C07285=1051.571,276.909,397.010,172.389,37.527,157.091
C07286=1051.565,276.657,397.040,172.386,37.524,157.091
C07287=1051.558,276.407,397.072,172.382,37.520,157.090
C07288=1051.551,276.156,397.102,172.380,37.518,157.089
C07289=1051.545,275.908,397.133,172.377,37.514,157.088
C07290=1051.539,275.660,397.164,172.374,37.511,157.088
C07291=1051.533,275.412,397.195,172.371,37.508,157.087
C07292=1051.526,275.164,397.225,172.368,37.504,157.086
C07293=1051.519,274.916,397.255,172.365,37.501,157.085
C07294=1051.513,274.668,397.286,172.363,37.498,157.085
C07295=1051.507,274.419,397.316,172.359,37.494,157.084
C07296=1051.500,274.172,397.347,172.357,37.491,157.083
C07297=1051.494,273.924,397.378,172.354,37.488,157.082
C07298=1051.487,273.675,397.408,172.350,37.485,157.082
C07299=1051.481,273.428,397.438,172.348,37.482,157.081
C07300=1051.474,273.179,397.469,172.345,37.478,157.080
C07301=1051.468,272.932,397.499,172.342,37.475,157.079
C07302=1051.461,272.683,397.529,172.339,37.472,157.079
C07303=1051.455,272.436,397.560,172.337,37.468,157.078
C07304=1051.449,272.187,397.590,172.333,37.465,157.077
C07305=1051.442,271.939,397.620,172.331,37.462,157.077
C07306=1051.436,271.691,397.651,172.328,37.458,157.076
C07307=1051.429,271.443,397.681,172.325,37.456,157.075
C07308=1051.423,271.195,397.711,172.322,37.452,157.074
C07309=1051.416,270.947,397.741,172.320,37.449,157.074
C07310=1051.410,270.699,397.772,172.317,37.446,157.073
C07311=1051.403,270.451,397.802,172.313,37.442,157.072
C07312=1051.397,270.203,397.832,172.311,37.439,157.071
C07313=1051.390,269.955,397.862,172.308,37.436,157.071
C07314=1051.384,269.707,397.893,172.305,37.433,157.070
C07315=1051.377,269.459,397.923,172.302,37.429,157.069
C07316=1051.371,269.210,397.952,172.300,37.427,157.069
C07317=1051.364,268.962,397.983,172.297,37.423,157.068
C07318=1051.358,268.714,398.013,172.294,37.420,157.067
C07319=1051.352,268.467,398.043,172.291,37.417,157.066
C07320=1051.346,268.218,398.073,172.289,37.413,157.066
C07321=1051.339,267.970,398.102,172.285,37.410,157.065
C07322=1051.332,267.722,398.133,172.283,37.407,157.064
C07323=1051.326,267.474,398.163,172.280,37.404,157.064
C07324=1051.319,267.226,398.193,172.278,37.400,157.063
C07325=1051.314,266.977,398.223,172.274,37.398,157.062
C07326=1051.306,266.729,398.253,172.272,37.394,157.061
C07327=1051.300,266.482,398.283,172.269,37.391,157.061
C07328=1051.294,266.232,398.313,172.267,37.388,157.060
C07329=1051.287,265.985,398.342,172.263,37.385,157.059
C07330=1051.281,265.737,398.372,172.261,37.381,157.058
C07331=1051.275,265.488,398.402,172.258,37.378,157.058
C07332=1051.268,265.241,398.432,172.256,37.375,157.057
C07333=1051.261,264.993,398.462,172.252,37.372,157.056
C07334=1051.255,264.744,398.492,172.250,37.368,157.056
C07335=1051.249,264.497,398.521,172.247,37.365,157.055
C07336=1051.242,264.248,398.551,172.244,37.362,157.054
C07337=1051.236,264.001,398.580,172.242,37.359,157.053
C07338=1051.229,263.753,398.610,172.238,37.356,157.053
C07339=1051.223,263.506,398.640,172.236,37.352,157.052
C07340=1051.216,263.258,398.669,172.233,37.349,157.051
C07341=1051.210,263.012,398.699,172.231,37.346,157.050
C07342=1051.204,262.764,398.729,172.228,37.343,157.050
C07343=1051.197,262.517,398.758,172.225,37.340,157.049
C07344=1051.191,262.269,398.788,172.222,37.336,157.048
C07345=1051.184,262.021,398.817,172.220,37.333,157.048
C07346=1051.178,261.772,398.846,172.217,37.330,157.047
C07347=1051.171,261.525,398.876,172.215,37.327,157.046
C07348=1051.165,261.277,398.905,172.211,37.324,157.046
C07349=1051.158,261.028,398.935,172.209,37.321,157.045
C07350=1051.151,260.780,398.964,172.206,37.318,157.044
C07351=1051.145,260.532,398.993,172.204,37.315,157.044
C07352=1051.138,260.283,399.023,172.201,37.311,157.043
C07353=1051.132,260.036,399.053,172.198,37.308,157.042
C07354=1051.125,259.787,399.082,172.196,37.305,157.042
C07355=1051.119,259.539,399.111,172.193,37.302,157.041
C07356=1051.112,259.291,399.141,172.191,37.299,157.040
C07357=1051.105,259.042,399.170,172.188,37.295,157.039
C07358=1051.099,258.794,399.199,172.184,37.293,157.039
C07359=1051.093,258.546,399.228,172.182,37.290,157.038
C07360=1051.086,258.298,399.257,172.179,37.286,157.037
C07361=1051.079,258.050,399.287,172.177,37.283,157.037
C07362=1051.072,257.802,399.316,172.175,37.280,157.036
C07363=1051.066,257.554,399.345,172.172,37.277,157.035
C07364=1051.059,257.305,399.374,172.170,37.274,157.035
C07365=1051.053,257.057,399.403,172.166,37.270,157.034
C07366=1051.047,256.809,399.432,172.164,37.267,157.033
C07367=1051.040,256.561,399.462,172.161,37.264,157.032
C07368=1051.033,256.312,399.492,172.159,37.261,157.032
C07369=1051.027,256.064,399.521,172.156,37.258,157.031
C07370=1051.021,255.816,399.550,172.154,37.255,157.030
C07371=1051.015,255.568,399.579,172.151,37.252,157.030
C07372=1051.008,255.319,399.608,172.148,37.249,157.029
C07373=1051.001,255.071,399.637,172.145,37.245,157.028
C07374=1050.995,254.823,399.666,172.143,37.242,157.028
C07375=1050.988,254.575,399.695,172.140,37.239,157.027
C07376=1050.982,254.327,399.724,172.138,37.236,157.026
C07377=1050.976,254.093,399.751,172.135,37.233,157.026
C07378=1050.970,253.860,399.779,172.133,37.230,157.025
C07379=1050.964,253.626,399.806,172.130,37.227,157.024
C07380=1050.958,253.392,399.833,172.128,37.223,157.023
C07381=1050.952,253.158,399.861,172.125,37.221,157.023
C07382=1050.946,252.925,399.888,172.123,37.218,157.022
C07383=1050.940,252.692,399.915,172.120,37.215,157.022
C07384=1050.934,252.458,399.943,172.118,37.212,157.021
C07385=1050.928,252.210,399.972,172.116,37.209,157.020
C07386=1050.920,251.962,400.001,172.113,37.205,157.019
C07387=1050.914,251.713,400.029,172.111,37.202,157.019
C07388=1050.908,251.465,400.058,172.108,37.199,157.018
C07389=1050.902,251.217,400.087,172.106,37.196,157.017
C07390=1050.896,250.969,400.116,172.103,37.192,157.017
C07391=1050.889,250.720,400.145,172.101,37.189,157.016
C07392=1050.883,250.472,400.174,172.098,37.186,157.015
C07393=1050.877,250.224,400.203,172.096,37.183,157.015
C07394=1050.871,249.975,400.232,172.093,37.180,157.014
C07395=1050.864,249.728,400.260,172.091,37.176,157.013
C07396=1050.858,249.479,400.289,172.088,37.174,157.013
C07397=1050.851,249.201,400.322,172.085,37.169,157.012
C07398=1050.843,248.924,400.354,172.082,37.166,157.011
C07399=1050.837,248.646,400.386,172.079,37.162,157.010
C07400=1050.830,248.368,400.418,172.077,37.159,157.009
C07401=1050.823,248.121,400.447,172.075,37.156,157.009
C07402=1050.817,247.872,400.475,172.072,37.152,157.008
C07403=1050.810,247.624,400.504,172.070,37.149,157.007
C07404=1050.804,247.376,400.533,172.067,37.146,157.006
C07405=1050.798,247.127,400.562,172.065,37.143,157.006
C07406=1050.792,246.879,400.591,172.062,37.139,157.005
C07407=1050.786,246.631,400.620,172.060,37.136,157.004
C07408=1050.779,246.382,400.647,172.057,37.133,157.004
C07409=1050.773,246.134,400.677,172.055,37.130,157.003
C07410=1050.767,245.886,400.706,172.052,37.126,157.002
C07411=1050.761,245.637,400.734,172.050,37.123,157.002
C07412=1050.754,245.389,400.762,172.047,37.120,157.001
C07413=1050.748,245.141,400.791,172.045,37.117,157.000
C07414=1050.741,244.892,400.820,172.042,37.114,157.000
C07415=1050.735,244.644,400.847,172.040,37.111,156.999
C07416=1050.729,244.396,400.876,172.037,37.108,156.998
C07417=1050.722,244.147,400.904,172.035,37.104,156.997
C07418=1050.716,243.899,400.933,172.032,37.101,156.997
C07419=1050.710,243.651,400.962,172.030,37.098,156.996
C07420=1050.703,243.403,400.990,172.027,37.095,156.995
C07421=1050.697,243.155,401.018,172.025,37.092,156.995
C07422=1050.690,242.907,401.046,172.022,37.088,156.994
C07423=1050.684,242.658,401.075,172.020,37.085,156.993
C07424=1050.678,242.409,401.103,172.017,37.082,156.993
C07425=1050.671,242.162,401.131,172.015,37.079,156.992
C07426=1050.666,241.913,401.160,172.013,37.076,156.991
C07427=1050.659,241.665,401.188,172.010,37.072,156.990
C07428=1050.653,241.416,401.217,172.008,37.069,156.990
C07429=1050.646,241.168,401.244,172.005,37.066,156.989
C07430=1050.639,240.920,401.273,172.003,37.063,156.988
C07431=1050.633,240.671,401.301,172.000,37.060,156.988
C07432=1050.626,240.423,401.329,171.999,37.056,156.987
C07433=1050.620,240.174,401.357,171.996,37.053,156.986
C07434=1050.613,239.926,401.386,171.994,37.050,156.986
C07435=1050.607,239.678,401.413,171.991,37.047,156.985
C07436=1050.601,239.429,401.442,171.989,37.044,156.984
C07437=1050.595,239.181,401.469,171.987,37.041,156.984
C07438=1050.588,238.933,401.497,171.984,37.037,156.983
C07439=1050.582,238.685,401.526,171.982,37.034,156.982
C07440=1050.575,238.436,401.554,171.979,37.031,156.982
C07441=1050.568,238.188,401.581,171.977,37.028,156.981
C07442=1050.562,237.939,401.610,171.974,37.025,156.980
C07443=1050.556,237.691,401.637,171.972,37.021,156.980
C07444=1050.549,237.442,401.665,171.969,37.018,156.979
C07445=1050.542,237.194,401.693,171.968,37.015,156.978
C07446=1050.537,236.946,401.721,171.965,37.012,156.977
C07447=1050.530,236.698,401.749,171.963,37.009,156.977
C07448=1050.523,236.449,401.777,171.961,37.006,156.976
C07449=1050.517,236.201,401.805,171.958,37.002,156.975
C07450=1050.511,235.952,401.833,171.956,36.999,156.975
C07451=1050.504,235.704,401.861,171.953,36.996,156.974
C07452=1050.497,235.455,401.888,171.951,36.993,156.973
C07453=1050.491,235.201,401.917,171.948,36.990,156.973
C07454=1050.485,234.947,401.945,171.946,36.986,156.972
C07455=1050.478,234.694,401.974,171.944,36.983,156.971
C07456=1050.472,234.439,402.003,171.942,36.980,156.971
C07457=1050.465,234.191,402.030,171.939,36.977,156.970
C07458=1050.459,233.943,402.058,171.937,36.973,156.969
C07459=1050.453,233.694,402.086,171.934,36.970,156.969
C07460=1050.447,233.446,402.114,171.932,36.967,156.968
C07461=1050.440,233.198,402.141,171.930,36.964,156.967
C07462=1050.433,232.949,402.169,171.928,36.960,156.966
C07463=1050.427,232.700,402.196,171.926,36.957,156.966
C07464=1050.422,232.452,402.224,171.923,36.954,156.965
C07465=1050.415,232.204,402.252,171.921,36.951,156.964
C07466=1050.408,231.955,402.280,171.918,36.948,156.964
C07467=1050.402,231.707,402.307,171.916,36.944,156.963
C07468=1050.395,231.458,402.335,171.913,36.941,156.962
C07469=1050.389,231.211,402.362,171.912,36.938,156.962
C07470=1050.383,230.962,402.389,171.909,36.935,156.961
C07471=1050.377,230.713,402.418,171.907,36.932,156.960
C07472=1050.371,230.465,402.445,171.904,36.928,156.960
C07473=1050.364,230.217,402.473,171.902,36.925,156.959
C07474=1050.357,229.968,402.501,171.901,36.922,156.958
C07475=1050.351,229.719,402.528,171.898,36.919,156.958
C07476=1050.345,229.471,402.555,171.896,36.916,156.957
C07477=1050.338,229.223,402.583,171.893,36.912,156.956
C07478=1050.331,228.974,402.610,171.891,36.909,156.956
C07479=1050.325,228.725,402.637,171.889,36.906,156.955
C07480=1050.319,228.478,402.665,171.887,36.903,156.954
C07481=1050.312,228.229,402.693,171.885,36.900,156.954
C07482=1050.306,227.980,402.720,171.882,36.897,156.953
C07483=1050.300,227.732,402.747,171.880,36.893,156.952
C07484=1050.293,227.483,402.774,171.877,36.890,156.951
C07485=1050.286,227.235,402.801,171.876,36.887,156.951
C07486=1050.279,226.987,402.829,171.873,36.884,156.950
C07487=1050.273,226.738,402.855,171.871,36.881,156.949
C07488=1050.267,226.490,402.883,171.868,36.877,156.949
C07489=1050.260,226.241,402.910,171.867,36.874,156.948
C07490=1050.254,225.993,402.938,171.865,36.871,156.947
C07491=1050.248,225.745,402.965,171.862,36.868,156.947
C07492=1050.241,225.496,402.992,171.860,36.865,156.946
C07493=1050.235,225.248,403.020,171.857,36.862,156.945
C07494=1050.228,224.999,403.046,171.856,36.858,156.945
C07495=1050.221,224.751,403.074,171.853,36.855,156.944
C07496=1050.216,224.502,403.100,171.851,36.852,156.943
C07497=1050.209,224.254,403.128,171.848,36.849,156.943
C07498=1050.203,224.006,403.155,171.847,36.846,156.942
C07499=1050.197,223.757,403.183,171.845,36.842,156.941
C07500=1050.190,223.508,403.210,171.842,36.839,156.941
C07501=1050.184,223.260,403.236,171.840,36.836,156.940
C07502=1050.177,223.012,403.263,171.838,36.833,156.939
C07503=1050.171,222.763,403.290,171.836,36.829,156.939
C07504=1050.164,222.515,403.318,171.833,36.826,156.938
C07505=1050.158,222.266,403.345,171.831,36.823,156.937
C07506=1050.152,222.018,403.372,171.830,36.819,156.937
C07507=1050.146,221.769,403.399,171.827,36.816,156.936
C07508=1050.139,221.521,403.425,171.825,36.813,156.935
C07509=1050.132,221.259,403.455,171.823,36.809,156.934
C07510=1050.126,220.997,403.483,171.821,36.806,156.934
C07511=1050.119,220.736,403.511,171.818,36.803,156.933
C07512=1050.113,220.474,403.540,171.816,36.799,156.932
C07513=1050.105,220.226,403.567,171.813,36.796,156.932
C07514=1050.099,219.977,403.593,171.812,36.793,156.931
C07515=1050.092,219.729,403.620,171.809,36.790,156.930
C07516=1050.087,219.480,403.646,171.807,36.787,156.930
C07517=1050.080,219.232,403.674,171.806,36.783,156.929
C07518=1050.073,218.984,403.700,171.803,36.780,156.928
C07519=1050.067,218.735,403.727,171.801,36.777,156.927
C07520=1050.060,218.486,403.754,171.798,36.774,156.927
C07521=1050.054,218.238,403.780,171.797,36.771,156.926
C07522=1050.047,217.989,403.808,171.794,36.767,156.925
C07523=1050.041,217.741,403.834,171.792,36.764,156.925
C07524=1050.035,217.492,403.861,171.791,36.760,156.924
C07525=1050.028,217.244,403.887,171.788,36.757,156.923
C07526=1050.022,216.995,403.914,171.786,36.754,156.923
C07527=1050.015,216.747,403.940,171.784,36.751,156.922
C07528=1050.009,216.498,403.967,171.782,36.748,156.921
C07529=1050.003,216.250,403.995,171.779,36.744,156.921
C07530=1049.996,216.001,404.021,171.778,36.741,156.920
C07531=1049.990,215.753,404.048,171.776,36.738,156.919
C07532=1049.983,215.504,404.074,171.773,36.735,156.919
C07533=1049.977,215.256,404.101,171.772,36.731,156.918
C07534=1049.970,215.007,404.127,171.769,36.728,156.917
C07535=1049.964,214.759,404.154,171.767,36.725,156.917
C07536=1049.958,214.510,404.180,171.765,36.722,156.916
C07537=1049.951,214.262,404.207,171.763,36.719,156.915
C07538=1049.945,214.013,404.233,171.761,36.715,156.915
C07539=1049.938,213.765,404.260,171.759,36.712,156.914
C07540=1049.932,213.516,404.287,171.757,36.708,156.913
C07541=1049.925,213.267,404.313,171.755,36.705,156.913
C07542=1049.920,213.019,404.340,171.753,36.702,156.912
C07543=1049.913,212.771,404.366,171.750,36.699,156.911
C07544=1049.907,212.522,404.393,171.749,36.695,156.910
C07545=1049.900,212.274,404.419,171.747,36.692,156.910
C07546=1049.894,212.025,404.446,171.744,36.689,156.909
C07547=1049.887,211.777,404.472,171.743,36.686,156.908
C07548=1049.881,211.528,404.499,171.740,36.682,156.908
C07549=1049.874,211.280,404.525,171.739,36.679,156.907
C07550=1049.868,211.031,404.550,171.736,36.675,156.906
C07551=1049.862,210.782,404.577,171.734,36.672,156.906
C07552=1049.855,210.534,404.603,171.733,36.669,156.905
C07553=1049.849,210.285,404.630,171.730,36.666,156.904
C07554=1049.842,210.037,404.656,171.729,36.662,156.904
C07555=1049.836,209.789,404.682,171.726,36.659,156.903
C07556=1049.830,209.539,404.709,171.724,36.656,156.902
C07557=1049.823,209.291,404.735,171.723,36.653,156.902
C07558=1049.817,209.043,404.761,171.720,36.649,156.901
C07559=1049.810,208.794,404.788,171.719,36.646,156.900
C07560=1049.804,208.546,404.814,171.716,36.643,156.899
C07561=1049.797,208.297,404.840,171.714,36.640,156.899
C07562=1049.791,208.049,404.866,171.712,36.636,156.898
C07563=1049.785,207.800,404.892,171.710,36.633,156.897
C07564=1049.778,207.551,404.919,171.709,36.629,156.897
C07565=1049.771,207.295,404.945,171.706,36.626,156.896
C07566=1049.765,207.039,404.972,171.704,36.623,156.895
C07567=1049.758,206.783,404.999,171.702,36.619,156.895
C07568=1049.752,206.527,405.026,171.700,36.616,156.894
C07569=1049.726,205.475,405.131,171.467,36.519,156.874
C07570=1049.720,205.226,405.157,171.464,36.516,156.873
C07571=1049.714,204.977,405.182,171.462,36.514,156.873
C07572=1049.707,204.729,405.207,171.460,36.512,156.872
C07573=1049.702,204.480,405.232,171.457,36.509,156.872
C07574=1049.695,204.232,405.256,171.454,36.507,156.871
C07575=1049.689,203.983,405.282,171.452,36.504,156.871
C07576=1049.683,203.734,405.306,171.449,36.501,156.870
C07577=1049.677,203.485,405.332,171.446,36.499,156.870
C07578=1049.671,203.237,405.357,171.444,36.497,156.869
C07579=1049.665,202.988,405.381,171.442,36.494,156.869
C07580=1049.659,202.739,405.407,171.438,36.492,156.868
C07581=1049.654,202.491,405.432,171.436,36.489,156.868
C07582=1049.648,202.242,405.456,171.434,36.487,156.867
C07583=1049.641,201.993,405.482,171.431,36.484,156.867
C07584=1049.636,201.744,405.506,171.428,36.482,156.866
C07585=1049.629,201.496,405.531,171.426,36.480,156.866
C07586=1049.623,201.247,405.555,171.424,36.477,156.865
C07587=1049.617,200.998,405.581,171.420,36.475,156.865
C07588=1049.610,200.749,405.605,171.418,36.472,156.864
C07589=1049.604,200.501,405.630,171.416,36.470,156.864
C07590=1049.599,200.252,405.654,171.413,36.467,156.863
C07591=1049.592,200.004,405.679,171.410,36.465,156.863
C07592=1049.586,199.755,405.704,171.408,36.463,156.862
C07593=1049.579,199.506,405.728,171.406,36.460,156.862
C07594=1049.574,199.258,405.753,171.403,36.458,156.861
C07595=1049.567,199.009,405.777,171.400,36.456,156.861
C07596=1049.561,198.760,405.802,171.398,36.454,156.861
C07597=1049.556,198.511,405.826,171.396,36.451,156.860
C07598=1049.549,198.263,405.851,171.392,36.449,156.860
C07599=1049.543,198.014,405.875,171.390,36.446,156.859
C07600=1049.537,197.765,405.899,171.388,36.444,156.859
C07601=1049.531,197.517,405.924,171.385,36.441,156.858
C07602=1049.525,197.267,405.949,171.383,36.439,156.858
C07603=1049.518,197.018,405.973,171.380,36.437,156.857
C07604=1049.512,196.771,405.998,171.378,36.435,156.857
C07605=1049.506,196.522,406.022,171.375,36.432,156.856
C07606=1049.501,196.273,406.046,171.373,36.430,156.856
C07607=1049.494,196.025,406.071,171.370,36.427,156.855
C07608=1049.488,195.775,406.096,171.367,36.425,156.855
C07609=1049.482,195.527,406.119,171.365,36.423,156.854
C07610=1049.476,195.278,406.144,171.363,36.421,156.854
C07611=1049.470,195.029,406.169,171.361,36.418,156.853
C07612=1049.464,194.781,406.193,171.357,36.416,156.853
C07613=1049.458,194.532,406.218,171.355,36.413,156.852
C07614=1049.452,194.283,406.241,171.353,36.411,156.852
C07615=1049.446,194.034,406.266,171.351,36.409,156.851
C07616=1049.439,193.786,406.291,171.348,36.407,156.851
C07617=1049.433,193.537,406.315,171.345,36.404,156.851
C07618=1049.427,193.288,406.339,171.343,36.402,156.850
C07619=1049.422,193.039,406.363,171.340,36.399,156.850
C07620=1049.415,192.790,406.387,171.338,36.397,156.849
C07621=1049.410,192.542,406.412,171.336,36.395,156.849
C07622=1049.403,192.293,406.436,171.333,36.393,156.848
C07623=1049.397,192.044,406.461,171.330,36.390,156.848
C07624=1049.391,191.796,406.485,171.328,36.388,156.847
C07625=1049.385,191.547,406.509,171.326,36.385,156.847
C07626=1049.379,191.298,406.533,171.324,36.384,156.846
C07627=1049.373,191.049,406.557,171.321,36.381,156.846
C07628=1049.368,190.801,406.582,171.318,36.379,156.846
C07629=1049.361,190.552,406.606,171.316,36.376,156.845
C07630=1049.354,190.267,406.633,171.314,36.374,156.845
C07631=1049.347,189.983,406.661,171.310,36.371,156.844
C07632=1049.341,189.699,406.688,171.308,36.368,156.843
C07633=1049.334,189.414,406.716,171.305,36.366,156.843
C07634=1049.328,189.166,406.740,171.302,36.364,156.842
C07635=1049.322,188.917,406.765,171.300,36.361,156.842
C07636=1049.316,188.669,406.788,171.298,36.359,156.842
C07637=1049.310,188.419,406.813,171.296,36.357,156.841
C07638=1049.304,188.171,406.837,171.293,36.354,156.841
C07639=1049.299,187.921,406.861,171.291,36.352,156.840
C07640=1049.292,187.673,406.884,171.289,36.350,156.840
C07641=1049.287,187.424,406.909,171.286,36.348,156.839
C07642=1049.281,187.175,406.933,171.283,36.345,156.839
C07643=1049.275,186.927,406.957,171.281,36.343,156.838
C07644=1049.269,186.678,406.981,171.279,36.340,156.838
C07645=1049.263,186.429,407.005,171.276,36.339,156.837
C07646=1049.257,186.180,407.029,171.274,36.336,156.837
C07647=1049.251,185.932,407.053,171.272,36.334,156.836
C07648=1049.246,185.683,407.076,171.270,36.331,156.836
C07649=1049.239,185.434,407.100,171.267,36.329,156.836
C07650=1049.234,185.185,407.125,171.264,36.327,156.835
C07651=1049.228,184.937,407.148,171.262,36.324,156.835
C07652=1049.222,184.688,407.173,171.260,36.322,156.834
C07653=1049.216,184.439,407.197,171.257,36.320,156.834
C07654=1049.211,184.190,407.220,171.255,36.318,156.833
C07655=1049.204,183.941,407.244,171.253,36.315,156.833
C07656=1049.198,183.693,407.268,171.251,36.313,156.832
C07657=1049.192,183.443,407.291,171.248,36.311,156.832
C07658=1049.186,183.195,407.315,171.246,36.309,156.832
C07659=1049.179,182.946,407.339,171.244,36.307,156.831
C07660=1049.173,182.697,407.362,171.241,36.305,156.831
C07661=1049.167,182.448,407.386,171.238,36.303,156.830
C07662=1049.161,182.199,407.409,171.236,36.301,156.830
C07663=1049.155,181.951,407.432,171.234,36.299,156.830
C07664=1049.148,181.702,407.456,171.232,36.296,156.829
C07665=1049.143,181.453,407.479,171.230,36.295,156.829
C07666=1049.135,181.204,407.503,171.227,36.292,156.828
C07667=1049.129,180.956,407.526,171.225,36.290,156.828
C07668=1049.123,180.707,407.550,171.223,36.288,156.828
C07669=1049.117,180.458,407.573,171.220,36.286,156.827
C07670=1049.111,180.209,407.596,171.217,36.284,156.827
C07671=1049.105,179.960,407.620,171.215,36.282,156.826
C07672=1049.099,179.711,407.643,171.213,36.280,156.826
C07673=1049.093,179.463,407.666,171.211,36.277,156.825
C07674=1049.086,179.214,407.690,171.208,36.276,156.825
C07675=1049.081,178.965,407.713,171.206,36.274,156.825
C07676=1049.074,178.716,407.737,171.204,36.271,156.824
C07677=1049.068,178.467,407.760,171.202,36.269,156.824
C07678=1049.062,178.219,407.784,171.199,36.267,156.823
C07679=1049.055,177.969,407.807,171.197,36.265,156.823
C07680=1049.049,177.720,407.830,171.195,36.263,156.822
C07681=1049.043,177.472,407.853,171.192,36.261,156.822
C07682=1049.038,177.223,407.876,171.190,36.259,156.822
C07683=1049.031,176.974,407.900,171.187,36.257,156.821
C07684=1049.025,176.725,407.923,171.185,36.255,156.821
C07685=1049.020,176.476,407.946,171.183,36.252,156.820
C07686=1049.013,176.227,407.970,171.181,36.250,156.820
C07687=1049.007,175.979,407.993,171.178,36.249,156.820
C07688=1049.000,175.731,408.016,171.176,36.246,156.819
C07689=1048.994,175.481,408.039,171.174,36.244,156.819
C07690=1048.988,175.232,408.062,171.172,36.242,156.818
C07691=1048.983,174.983,408.085,171.170,36.240,156.818
C07692=1048.977,174.735,408.109,171.167,36.238,156.818
C07693=1048.970,174.485,408.132,171.165,36.236,156.817
C07694=1048.963,174.201,408.158,171.163,36.233,156.817
C07695=1048.956,173.916,408.185,171.160,36.231,156.816
C07696=1048.950,173.631,408.212,171.157,36.229,156.816
C07697=1048.942,173.347,408.238,171.155,36.226,156.815
C07698=1048.937,173.098,408.261,171.153,36.224,156.815
C07699=1048.931,172.849,408.284,171.151,36.222,156.814
C07700=1048.925,172.600,408.307,171.148,36.220,156.814
C07701=1048.918,172.351,408.331,171.146,36.218,156.814
C07702=1048.912,172.102,408.354,171.144,36.216,156.813
C07703=1048.906,171.854,408.377,171.142,36.214,156.813
C07704=1048.901,171.605,408.399,171.139,36.212,156.812
C07705=1048.895,171.356,408.422,171.137,36.210,156.812
C07706=1048.889,171.107,408.445,171.135,36.207,156.812
C07707=1048.882,170.858,408.469,171.133,36.206,156.811
C07708=1048.876,170.609,408.492,171.131,36.203,156.811
C07709=1048.870,170.360,408.515,171.128,36.201,156.810
C07710=1048.865,170.112,408.538,171.126,36.199,156.810
C07711=1048.859,169.863,408.561,171.124,36.197,156.810
C07712=1048.853,169.614,408.584,171.122,36.195,156.809
C07713=1048.847,169.365,408.606,171.119,36.193,156.809
C07714=1048.840,169.116,408.629,171.117,36.191,156.808
C07715=1048.834,168.867,408.653,171.115,36.189,156.808
C07716=1048.829,168.618,408.676,171.113,36.187,156.807
C07717=1048.823,168.369,408.699,171.111,36.185,156.807
C07718=1048.817,168.121,408.722,171.108,36.183,156.807
C07719=1048.811,167.872,408.745,171.106,36.180,156.806
C07720=1048.805,167.623,408.767,171.104,36.179,156.806
C07721=1048.799,167.374,408.790,171.102,36.176,156.805
C07722=1048.793,167.125,408.813,171.099,36.174,156.805
C07723=1048.788,166.876,408.836,171.097,36.172,156.805
C07724=1048.782,166.627,408.859,171.095,36.170,156.804
C07725=1048.775,166.379,408.881,171.093,36.168,156.804
C07726=1048.769,166.129,408.904,171.091,36.166,156.804
C07727=1048.763,165.880,408.927,171.088,36.164,156.803
C07728=1048.758,165.632,408.950,171.086,36.162,156.803
C07729=1048.752,165.383,408.973,171.084,36.159,156.802
C07730=1048.745,165.134,408.996,171.082,36.158,156.802
C07731=1048.740,164.885,409.019,171.079,36.156,156.801
C07732=1048.734,164.636,409.041,171.077,36.153,156.801
C07733=1048.729,164.387,409.064,171.076,36.151,156.801
C07734=1048.723,164.138,409.087,171.074,36.150,156.800
C07735=1048.716,163.889,409.109,171.072,36.147,156.800
C07736=1048.711,163.640,409.132,171.069,36.145,156.799
C07737=1048.705,163.391,409.155,171.067,36.143,156.799
C07738=1048.699,163.143,409.178,171.065,36.141,156.799
C07739=1048.693,162.894,409.200,171.063,36.139,156.798
C07740=1048.687,162.644,409.222,171.060,36.137,156.798
C07741=1048.682,162.396,409.245,171.058,36.135,156.797
C07742=1048.676,162.147,409.268,171.056,36.133,156.797
C07743=1048.669,161.898,409.291,171.054,36.130,156.797
C07744=1048.664,161.650,409.313,171.053,36.129,156.796
C07745=1048.658,161.401,409.336,171.050,36.127,156.796
C07746=1048.653,161.151,409.358,171.048,36.124,156.795
C07747=1048.647,160.903,409.381,171.046,36.122,156.795
C07748=1048.641,160.654,409.404,171.044,36.120,156.795
C07749=1048.635,160.405,409.427,171.042,36.118,156.794
C07750=1048.629,160.156,409.448,171.039,36.116,156.794
C07751=1048.623,159.907,409.471,171.037,36.114,156.793
C07752=1048.617,159.658,409.494,171.035,36.113,156.793
C07753=1048.611,159.409,409.515,171.033,36.111,156.793
C07754=1048.605,159.160,409.538,171.031,36.108,156.792
C07755=1048.599,158.911,409.560,171.028,36.106,156.792
C07756=1048.593,158.662,409.583,171.027,36.105,156.792
C07757=1048.587,158.414,409.605,171.025,36.103,156.791
C07758=1048.579,158.128,409.630,171.022,36.100,156.791
C07759=1048.572,157.843,409.656,171.020,36.098,156.790
C07760=1048.565,157.558,409.681,171.017,36.096,156.790
C07761=1048.559,157.272,409.706,171.015,36.094,156.790
C07762=1048.553,157.024,409.729,171.013,36.092,156.789
C07763=1048.547,156.774,409.751,171.011,36.090,156.789
C07764=1048.541,156.525,409.774,171.008,36.088,156.788
C07765=1048.535,156.277,409.796,171.006,36.086,156.788
C07766=1048.528,156.028,409.818,171.004,36.084,156.788
C07767=1048.523,155.779,409.841,171.003,36.082,156.787
C07768=1048.517,155.530,409.863,171.001,36.080,156.787
C07769=1048.510,155.281,409.885,170.998,36.078,156.786
C07770=1048.505,155.031,409.907,170.996,36.076,156.786
C07771=1048.498,154.783,409.929,170.994,36.074,156.786
C07772=1048.492,154.534,409.951,170.992,36.072,156.785
C07773=1048.486,154.285,409.974,170.990,36.070,156.785
C07774=1048.481,154.036,409.995,170.987,36.069,156.785
C07775=1048.475,153.787,410.017,170.985,36.067,156.784
C07776=1048.468,153.539,410.039,170.984,36.064,156.784
C07777=1048.462,153.289,410.061,170.982,36.062,156.783
C07778=1048.456,153.040,410.084,170.980,36.061,156.783
C07779=1048.450,152.791,410.106,170.977,36.059,156.783
C07780=1048.444,152.542,410.127,170.975,36.057,156.782
C07781=1048.437,152.293,410.149,170.973,36.055,156.782
C07782=1048.432,152.044,410.172,170.971,36.053,156.782
C07783=1048.426,151.795,410.193,170.969,36.051,156.781
C07784=1048.420,151.547,410.215,170.968,36.049,156.781
C07785=1048.414,151.298,410.237,170.965,36.048,156.781
C07786=1048.408,151.048,410.259,170.963,36.046,156.780
C07787=1048.402,150.799,410.282,170.961,36.043,156.780
C07788=1048.396,150.550,410.303,170.959,36.041,156.779
C07789=1048.390,150.301,410.325,170.957,36.039,156.779
C07790=1048.384,150.053,410.347,170.954,36.038,156.779
C07791=1048.378,149.804,410.368,170.953,36.036,156.778
C07792=1048.372,149.554,410.391,170.951,36.034,156.778
C07793=1048.366,149.306,410.413,170.949,36.032,156.778
C07794=1048.359,149.057,410.435,170.947,36.030,156.777
C07795=1048.354,148.808,410.456,170.944,36.028,156.777
C07796=1048.348,148.559,410.478,170.942,36.026,156.777
C07797=1048.342,148.310,410.499,170.941,36.025,156.776
C07798=1048.335,148.061,410.522,170.939,36.023,156.776
C07799=1048.329,147.812,410.543,170.937,36.021,156.775
C07800=1048.324,147.562,410.565,170.935,36.019,156.775
C07801=1048.318,147.314,410.587,170.932,36.017,156.775
C07802=1048.312,147.065,410.608,170.930,36.015,156.774
C07803=1048.305,146.816,410.631,170.928,36.013,156.774
C07804=1048.299,146.567,410.652,170.927,36.012,156.774
C07805=1048.293,146.318,410.674,170.925,36.010,156.773
C07806=1048.287,146.069,410.695,170.922,36.008,156.773
C07807=1048.281,145.820,410.716,170.920,36.006,156.773
C07808=1048.274,145.571,410.738,170.918,36.004,156.772
C07809=1048.268,145.322,410.760,170.916,36.002,156.772
C07810=1048.262,145.073,410.781,170.915,36.000,156.772
C07811=1048.257,144.824,410.802,170.913,35.998,156.771
C07812=1048.250,144.575,410.824,170.910,35.997,156.771
C07813=1048.244,144.326,410.846,170.908,35.995,156.771
C07814=1048.238,144.077,410.867,170.906,35.993,156.770
C07815=1048.232,143.829,410.889,170.904,35.991,156.770
C07816=1048.226,143.580,410.911,170.903,35.989,156.769
C07817=1048.220,143.330,410.933,170.900,35.987,156.769
C07818=1048.214,143.081,410.954,170.898,35.985,156.769
C07819=1048.208,142.833,410.976,170.896,35.984,156.768
C07820=1048.202,142.583,410.997,170.894,35.982,156.768
C07821=1048.196,142.334,411.019,170.893,35.980,156.768
C07822=1048.189,142.049,411.042,170.889,35.977,156.767
C07823=1048.182,141.763,411.068,170.887,35.975,156.767
C07824=1048.175,141.477,411.092,170.885,35.974,156.766
C07825=1048.168,141.193,411.116,170.883,35.971,156.766
C07826=1048.162,140.943,411.138,170.881,35.969,156.766
C07827=1048.156,140.694,411.160,170.879,35.967,156.765
C07828=1048.150,140.446,411.181,170.877,35.966,156.765
C07829=1048.144,140.196,411.203,170.875,35.964,156.765
C07830=1048.138,139.947,411.223,170.873,35.962,156.764
C07831=1048.133,139.698,411.245,170.872,35.960,156.764
C07832=1048.126,139.449,411.266,170.870,35.958,156.764
C07833=1048.120,139.200,411.288,170.867,35.956,156.763
C07834=1048.113,138.951,411.309,170.865,35.954,156.763
C07835=1048.108,138.702,411.330,170.863,35.952,156.762
C07836=1048.102,138.453,411.352,170.862,35.951,156.762
C07837=1048.096,138.203,411.373,170.860,35.949,156.762
C07838=1048.089,137.955,411.394,170.858,35.947,156.762
C07839=1048.083,137.706,411.415,170.855,35.946,156.761
C07840=1048.077,137.457,411.437,170.853,35.944,156.761
C07841=1048.072,137.208,411.458,170.852,35.942,156.760
C07842=1048.065,136.959,411.478,170.850,35.940,156.760
C07843=1048.059,136.709,411.500,170.848,35.938,156.760
C07844=1048.053,136.461,411.521,170.845,35.936,156.759
C07845=1048.047,136.211,411.542,170.843,35.934,156.759
C07846=1048.040,135.962,411.563,170.842,35.932,156.759
C07847=1048.035,135.714,411.585,170.840,35.931,156.758
C07848=1048.029,135.464,411.606,170.838,35.929,156.758
C07849=1048.023,135.216,411.626,170.836,35.927,156.758
C07850=1048.017,134.966,411.648,170.834,35.926,156.757
C07851=1048.010,134.717,411.669,170.832,35.924,156.757
C07852=1048.004,134.468,411.689,170.830,35.922,156.757
C07853=1047.998,134.219,411.711,170.828,35.920,156.756
C07854=1047.992,133.970,411.733,170.826,35.918,156.756
C07855=1047.986,133.721,411.753,170.825,35.916,156.756
C07856=1047.980,133.472,411.774,170.822,35.914,156.755
C07857=1047.974,133.224,411.796,170.820,35.913,156.755
C07858=1047.968,132.974,411.816,170.818,35.911,156.755
C07859=1047.962,132.726,411.837,170.817,35.909,156.754
C07860=1047.956,132.476,411.859,170.815,35.907,156.754
C07861=1047.949,132.227,411.879,170.813,35.906,156.754
C07862=1047.944,131.978,411.900,170.810,35.904,156.753
C07863=1047.938,131.728,411.921,170.809,35.902,156.753
C07864=1047.932,131.480,411.942,170.807,35.900,156.753
C07865=1047.926,131.230,411.963,170.805,35.898,156.752
C07866=1047.919,130.982,411.984,170.803,35.897,156.752
C07867=1047.914,130.732,412.004,170.802,35.895,156.752
C07868=1047.907,130.484,412.025,170.799,35.893,156.751
C07869=1047.901,130.235,412.045,170.797,35.891,156.751
C07870=1047.895,129.986,412.067,170.795,35.890,156.751
C07871=1047.888,129.736,412.087,170.793,35.888,156.750
C07872=1047.883,129.487,412.109,170.792,35.886,156.750
C07873=1047.876,129.238,412.129,170.790,35.884,156.750
C07874=1047.870,128.990,412.150,170.787,35.882,156.749
C07875=1047.864,128.740,412.171,170.785,35.881,156.749
C07876=1047.857,128.491,412.192,170.784,35.879,156.749
C07877=1047.851,128.242,412.212,170.782,35.877,156.748
C07878=1047.845,127.992,412.233,170.780,35.876,156.748
C07879=1047.839,127.744,412.253,170.778,35.874,156.748
C07880=1047.832,127.495,412.274,170.776,35.872,156.747
C07881=1047.827,127.246,412.295,170.774,35.871,156.747
C07882=1047.820,126.997,412.315,170.772,35.869,156.747
C07883=1047.815,126.748,412.336,170.770,35.867,156.746
C07884=1047.808,126.499,412.357,170.769,35.866,156.746
C07885=1047.801,126.249,412.377,170.767,35.864,156.746
C07886=1047.794,125.964,412.401,170.765,35.862,156.745
C07887=1047.787,125.678,412.424,170.762,35.860,156.745
C07888=1047.781,125.392,412.447,170.760,35.857,156.745
C07889=1047.773,125.106,412.471,170.758,35.855,156.744
C07890=1047.768,124.857,412.492,170.756,35.854,156.744
C07891=1047.761,124.608,412.513,170.754,35.852,156.744
C07892=1047.755,124.359,412.533,170.752,35.850,156.743
C07893=1047.749,124.110,412.553,170.750,35.849,156.743
C07894=1047.743,123.861,412.574,170.748,35.847,156.743
C07895=1047.737,123.613,412.594,170.746,35.845,156.742
C07896=1047.731,123.363,412.615,170.745,35.844,156.742
C07897=1047.725,123.114,412.635,170.743,35.842,156.742
C07898=1047.718,122.865,412.656,170.741,35.840,156.741
C07899=1047.713,122.616,412.677,170.739,35.838,156.741
C07900=1047.706,122.366,412.697,170.737,35.837,156.741
C07901=1047.700,122.118,412.717,170.735,35.835,156.740
C07902=1047.694,121.868,412.738,170.733,35.833,156.740
C07903=1047.688,121.620,412.759,170.732,35.831,156.740
C07904=1047.682,121.371,412.779,170.730,35.829,156.739
C07905=1047.676,121.121,412.800,170.727,35.828,156.739
C07906=1047.670,120.872,412.820,170.726,35.826,156.739
C07907=1047.663,120.623,412.840,170.724,35.824,156.738
C07908=1047.658,120.374,412.861,170.722,35.822,156.738
C07909=1047.652,120.125,412.881,170.720,35.820,156.738
C07910=1047.645,119.876,412.901,170.719,35.818,156.737
C07911=1047.639,119.627,412.921,170.716,35.817,156.737
C07912=1047.633,119.377,412.942,170.714,35.815,156.737
C07913=1047.627,119.128,412.962,170.713,35.813,156.736
C07914=1047.621,118.880,412.982,170.711,35.812,156.736
C07915=1047.616,118.630,413.003,170.709,35.810,156.736
C07916=1047.609,118.382,413.024,170.708,35.808,156.736
C07917=1047.603,118.132,413.044,170.706,35.807,156.735
C07918=1047.597,117.883,413.065,170.703,35.805,156.735
C07919=1047.591,117.634,413.085,170.701,35.803,156.734
C07920=1047.585,117.385,413.105,170.700,35.801,156.734
C07921=1047.579,117.136,413.125,170.698,35.799,156.734
C07922=1047.574,116.887,413.146,170.696,35.798,156.734
C07923=1047.567,116.637,413.166,170.695,35.796,156.733
C07924=1047.561,116.388,413.186,170.692,35.794,156.733
C07925=1047.555,116.139,413.206,170.690,35.792,156.732
C07926=1047.549,115.890,413.227,170.689,35.790,156.732
C07927=1047.543,115.641,413.247,170.687,35.788,156.732
C07928=1047.537,115.392,413.267,170.685,35.787,156.732
C07929=1047.532,115.143,413.287,170.684,35.785,156.731
C07930=1047.525,114.893,413.308,170.681,35.783,156.731
C07931=1047.519,114.645,413.327,170.679,35.781,156.731
C07932=1047.513,114.396,413.347,170.678,35.780,156.730
C07933=1047.507,114.146,413.368,170.676,35.778,156.730
C07934=1047.501,113.897,413.388,170.674,35.776,156.730
C07935=1047.495,113.648,413.408,170.673,35.774,156.729
C07936=1047.489,113.399,413.429,170.670,35.773,156.729
C07937=1047.483,113.150,413.449,170.668,35.771,156.729
C07938=1047.477,112.901,413.469,170.666,35.769,156.728
C07939=1047.471,112.651,413.488,170.665,35.768,156.728
C07940=1047.465,112.402,413.508,170.663,35.766,156.728
C07941=1047.459,112.153,413.528,170.661,35.764,156.727
C07942=1047.453,111.905,413.548,170.660,35.763,156.727
C07943=1047.446,111.655,413.568,170.657,35.761,156.727
C07944=1047.440,111.406,413.588,170.655,35.759,156.726
C07945=1047.434,111.157,413.608,170.654,35.757,156.726
C07946=1047.428,110.907,413.628,170.652,35.756,156.726
C07947=1047.422,110.658,413.648,170.650,35.754,156.725
C07948=1047.416,110.410,413.668,170.649,35.752,156.725
C07949=1047.409,110.160,413.688,170.647,35.751,156.725
C07950=1047.402,109.874,413.710,170.644,35.749,156.724
C07951=1047.395,109.588,413.733,170.642,35.747,156.724
C07952=1047.388,109.303,413.756,170.640,35.745,156.724
C07953=1047.381,109.017,413.779,170.638,35.743,156.723
C07954=1047.375,108.768,413.799,170.636,35.741,156.723
C07955=1047.369,108.518,413.818,170.635,35.739,156.723
C07956=1047.363,108.269,413.838,170.632,35.738,156.723
C07957=1047.356,108.020,413.858,170.630,35.736,156.722
C07958=1047.350,107.771,413.877,170.629,35.734,156.722
C07959=1047.344,107.522,413.897,170.627,35.733,156.722
C07960=1047.338,107.273,413.917,170.625,35.731,156.721
C07961=1047.332,107.024,413.937,170.624,35.729,156.721
C07962=1047.326,106.774,413.956,170.622,35.728,156.721
C07963=1047.320,106.526,413.976,170.619,35.726,156.720
C07964=1047.313,106.276,413.995,170.618,35.724,156.720
C07965=1047.307,106.027,414.015,170.616,35.723,156.720
C07966=1047.301,105.778,414.035,170.614,35.721,156.719
C07967=1047.295,105.529,414.054,170.613,35.719,156.719
C07968=1047.289,105.280,414.074,170.611,35.718,156.719
C07969=1047.283,105.030,414.095,170.609,35.716,156.718
C07970=1047.276,104.781,414.113,170.607,35.714,156.718
C07971=1047.270,104.532,414.133,170.605,35.712,156.718
C07972=1047.265,104.283,414.153,170.603,35.711,156.718
C07973=1047.259,104.034,414.173,170.602,35.709,156.717
C07974=1047.252,103.784,414.192,170.600,35.707,156.717
C07975=1047.246,103.535,414.212,170.598,35.706,156.717
C07976=1047.239,103.287,414.231,170.597,35.704,156.716
C07977=1047.234,103.037,414.251,170.594,35.702,156.716
C07978=1047.228,102.789,414.271,170.592,35.701,156.716
C07979=1047.222,102.539,414.290,170.591,35.699,156.715
C07980=1047.216,102.290,414.310,170.589,35.697,156.715
C07981=1047.209,102.040,414.329,170.587,35.695,156.715
C07982=1047.203,101.792,414.349,170.586,35.694,156.714
C07983=1047.197,101.542,414.368,170.584,35.692,156.714
C07984=1047.191,101.293,414.388,170.582,35.690,156.714
C07985=1047.186,101.044,414.407,170.580,35.689,156.713
C07986=1047.179,100.796,414.427,170.578,35.687,156.713
C07987=1047.173,100.545,414.446,170.577,35.685,156.713
C07988=1047.167,100.297,414.466,170.575,35.684,156.713
C07989=1047.160,100.047,414.485,170.573,35.682,156.712
C07990=1047.155,99.798,414.504,170.571,35.680,156.712
C07991=1047.148,99.549,414.523,170.569,35.679,156.712
C07992=1047.142,99.300,414.543,170.567,35.677,156.711
C07993=1047.136,99.051,414.563,170.566,35.675,156.711
C07994=1047.129,98.801,414.582,170.564,35.673,156.711
C07995=1047.123,98.552,414.601,170.562,35.672,156.711
C07996=1047.117,98.303,414.620,170.561,35.670,156.710
C07997=1047.111,98.054,414.640,170.559,35.668,156.710
C07998=1047.105,97.805,414.658,170.556,35.667,156.710
C07999=1047.099,97.556,414.678,170.555,35.665,156.709
C08000=1047.092,97.306,414.698,170.553,35.664,156.709
C08001=1047.086,97.057,414.716,170.551,35.662,156.709
C08002=1047.080,96.808,414.736,170.550,35.660,156.708
C08003=1047.074,96.559,414.755,170.548,35.659,156.708
C08004=1047.068,96.309,414.774,170.546,35.657,156.708
C08005=1047.061,96.060,414.793,170.544,35.656,156.708
C08006=1047.055,95.812,414.813,170.542,35.654,156.707
C08007=1047.049,95.562,414.831,170.540,35.652,156.707
C08008=1047.043,95.313,414.851,170.539,35.651,156.707
C08009=1047.037,95.064,414.869,170.537,35.649,156.706
C08010=1047.030,94.814,414.890,170.535,35.647,156.706
C08011=1047.024,94.565,414.908,170.534,35.646,156.706
C08012=1047.018,94.316,414.928,170.531,35.644,156.705
C08013=1047.012,94.066,414.947,170.529,35.642,156.705
C08014=1047.006,93.781,414.969,170.528,35.641,156.705
C08015=1046.998,93.495,414.990,170.526,35.639,156.704
C08016=1046.991,93.209,415.013,170.524,35.637,156.704
C08017=1046.984,92.923,415.034,170.522,35.634,156.704
C08018=1046.978,92.674,415.054,170.520,35.633,156.703
C08019=1046.972,92.425,415.073,170.518,35.631,156.703
C08020=1046.966,92.176,415.092,170.516,35.630,156.703
C08021=1046.959,91.927,415.111,170.514,35.628,156.702
C08022=1046.954,91.677,415.130,170.513,35.626,156.702
C08023=1046.947,91.428,415.149,170.511,35.625,156.702
C08024=1046.942,91.179,415.168,170.509,35.623,156.702
C08025=1046.935,90.930,415.187,170.508,35.621,156.701
C08026=1046.929,90.681,415.207,170.506,35.620,156.701
C08027=1046.923,90.431,415.225,170.504,35.618,156.701
C08028=1046.917,90.182,415.245,170.502,35.616,156.700
C08029=1046.911,89.933,415.263,170.500,35.614,156.700
C08030=1046.904,89.684,415.282,170.499,35.613,156.700
C08031=1046.898,89.435,415.300,170.497,35.611,156.699
C08032=1046.892,89.185,415.320,170.495,35.609,156.699
C08033=1046.886,88.936,415.338,170.494,35.608,156.699
C08034=1046.879,88.687,415.357,170.491,35.606,156.699
C08035=1046.873,88.438,415.376,170.489,35.605,156.698
C08036=1046.867,88.188,415.395,170.488,35.603,156.698
C08037=1046.861,87.939,415.414,170.486,35.602,156.698
C08038=1046.854,87.690,415.432,170.484,35.600,156.697
C08039=1046.848,87.441,415.451,170.483,35.599,156.697
C08040=1046.842,87.192,415.470,170.481,35.597,156.697
C08041=1046.836,86.943,415.489,170.479,35.595,156.697
C08042=1046.829,86.693,415.507,170.477,35.593,156.696
C08043=1046.823,86.444,415.526,170.475,35.592,156.696
C08044=1046.817,86.195,415.545,170.473,35.590,156.696
C08045=1046.811,85.946,415.564,170.472,35.589,156.695
C08046=1046.804,85.697,415.583,170.470,35.587,156.695
C08047=1046.798,85.448,415.601,170.469,35.586,156.695
C08048=1046.792,85.198,415.619,170.467,35.584,156.695
C08049=1046.786,84.948,415.638,170.464,35.582,156.694
C08050=1046.780,84.699,415.657,170.463,35.581,156.694
C08051=1046.773,84.450,415.676,170.461,35.579,156.694
C08052=1046.767,84.201,415.694,170.459,35.578,156.693
C08053=1046.761,83.952,415.714,170.458,35.576,156.693
C08054=1046.755,83.702,415.732,170.456,35.574,156.693
C08055=1046.748,83.453,415.751,170.454,35.572,156.693
C08056=1046.743,83.204,415.768,170.453,35.571,156.692
C08057=1046.736,82.955,415.787,170.450,35.569,156.692
C08058=1046.731,82.706,415.806,170.449,35.567,156.692
C08059=1046.724,82.457,415.825,170.447,35.566,156.691
C08060=1046.718,82.207,415.844,170.445,35.564,156.691
C08061=1046.711,81.958,415.862,170.444,35.563,156.691
C08062=1046.705,81.709,415.880,170.442,35.561,156.690
C08063=1046.700,81.459,415.900,170.440,35.560,156.690
C08064=1046.693,81.210,415.918,170.439,35.558,156.690
C08065=1046.687,80.961,415.937,170.436,35.557,156.690
C08066=1046.681,80.712,415.955,170.434,35.555,156.689
C08067=1046.675,80.463,415.973,170.433,35.553,156.689
C08068=1046.669,80.213,415.992,170.431,35.551,156.689
C08069=1046.663,79.964,416.011,170.430,35.550,156.688
C08070=1046.656,79.715,416.030,170.428,35.548,156.688
C08071=1046.650,79.465,416.047,170.426,35.546,156.688
C08072=1046.644,79.216,416.066,170.425,35.544,156.687
C08073=1046.639,78.967,416.085,170.422,35.543,156.687
C08074=1046.632,78.718,416.103,170.420,35.541,156.687
C08075=1046.626,78.469,416.122,170.419,35.540,156.687
C08076=1046.620,78.219,416.140,170.417,35.538,156.686
C08077=1046.614,77.970,416.158,170.416,35.537,156.686
C08078=1046.607,77.684,416.179,170.414,35.535,156.686
C08079=1046.599,77.398,416.200,170.412,35.533,156.685
C08080=1046.593,77.112,416.222,170.409,35.531,156.685
C08081=1046.585,76.826,416.243,170.407,35.529,156.685
C08082=1046.579,76.577,416.261,170.405,35.528,156.685
C08083=1046.573,76.328,416.279,170.404,35.526,156.684
C08084=1046.566,76.079,416.298,170.402,35.525,156.684
C08085=1046.560,75.829,416.316,170.400,35.523,156.684
C08086=1046.554,75.580,416.334,170.399,35.521,156.683
C08087=1046.548,75.331,416.352,170.397,35.520,156.683
C08088=1046.541,75.081,416.371,170.396,35.518,156.683
C08089=1046.536,74.832,416.388,170.393,35.516,156.682
C08090=1046.529,74.583,416.407,170.391,35.515,156.682
C08091=1046.523,74.334,416.426,170.390,35.513,156.682
C08092=1046.517,74.084,416.444,170.388,35.512,156.682
C08093=1046.510,73.836,416.462,170.386,35.511,156.681
C08094=1046.503,73.586,416.480,170.385,35.509,156.681
C08095=1046.498,73.337,416.498,170.383,35.507,156.681
C08096=1046.492,73.088,416.516,170.381,35.505,156.681
C08097=1046.485,72.839,416.534,170.379,35.504,156.680
C08098=1046.479,72.589,416.552,170.377,35.502,156.680
C08099=1046.473,72.340,416.571,170.375,35.501,156.680
C08100=1046.467,72.091,416.589,170.374,35.499,156.679
C08101=1046.461,71.842,416.607,170.372,35.498,156.679
C08102=1046.454,71.592,416.625,170.371,35.496,156.679
C08103=1046.448,71.342,416.643,170.369,35.495,156.679
C08104=1046.442,71.094,416.661,170.367,35.493,156.678
C08105=1046.436,70.844,416.679,170.365,35.491,156.678
C08106=1046.429,70.595,416.697,170.363,35.489,156.678
C08107=1046.423,70.345,416.715,170.361,35.488,156.678
C08108=1046.417,70.097,416.734,170.360,35.486,156.677
C08109=1046.411,69.847,416.752,170.358,35.485,156.677
C08110=1046.405,69.597,416.769,170.356,35.483,156.677
C08111=1046.399,69.348,416.788,170.355,35.482,156.676
C08112=1046.392,69.100,416.805,170.353,35.480,156.676
C08113=1046.386,68.850,416.823,170.351,35.479,156.676
C08114=1046.380,68.601,416.842,170.349,35.477,156.675
C08115=1046.374,68.351,416.860,170.347,35.475,156.675
C08116=1046.367,68.102,416.877,170.346,35.474,156.675
C08117=1046.361,67.853,416.895,170.344,35.472,156.675
C08118=1046.355,67.603,416.913,170.342,35.471,156.674
C08119=1046.349,67.354,416.931,170.341,35.469,156.674
C08120=1046.342,67.106,416.949,170.339,35.468,156.674
C08121=1046.336,66.856,416.967,170.337,35.466,156.674
C08122=1046.330,66.606,416.985,170.335,35.464,156.673
C08123=1046.324,66.357,417.002,170.333,35.463,156.673
C08124=1046.317,66.108,417.020,170.331,35.461,156.673
C08125=1046.311,65.859,417.038,170.330,35.460,156.673
C08126=1046.306,65.609,417.056,170.328,35.458,156.672
C08127=1046.299,65.360,417.073,170.327,35.457,156.672
C08128=1046.292,65.111,417.092,170.325,35.455,156.672
C08129=1046.286,64.861,417.110,170.323,35.454,156.671
C08130=1046.280,64.612,417.127,170.321,35.452,156.671
C08131=1046.274,64.363,417.145,170.319,35.450,156.671
C08132=1046.268,64.113,417.163,170.317,35.449,156.671
C08133=1046.261,63.865,417.180,170.316,35.447,156.670
C08134=1046.255,63.615,417.198,170.314,35.446,156.670
C08135=1046.248,63.366,417.215,170.312,35.445,156.670
C08136=1046.242,63.116,417.233,170.311,35.443,156.670
C08137=1046.236,62.867,417.250,170.309,35.441,156.669
C08138=1046.230,62.617,417.268,170.307,35.440,156.669
C08139=1046.223,62.368,417.286,170.305,35.438,156.669
C08140=1046.217,62.119,417.303,170.303,35.437,156.669
C08141=1046.210,61.870,417.321,170.301,35.436,156.668
C08142=1046.203,61.584,417.342,170.299,35.434,156.668
C08143=1046.196,61.298,417.362,170.297,35.432,156.668
C08144=1046.189,61.012,417.381,170.296,35.430,156.667
C08145=1046.180,60.725,417.401,170.294,35.428,156.667
C08146=1046.175,60.476,417.419,170.292,35.427,156.667
C08147=1046.168,60.227,417.436,170.290,35.426,156.667
C08148=1046.162,59.977,417.454,170.288,35.424,156.666
C08149=1046.156,59.728,417.471,170.286,35.423,156.666
C08150=1046.150,59.479,417.489,170.284,35.421,156.666
C08151=1046.143,59.229,417.506,170.283,35.419,156.665
C08152=1046.136,58.981,417.523,170.281,35.418,156.665
C08153=1046.130,58.731,417.541,170.279,35.417,156.665
C08154=1046.123,58.481,417.559,170.278,35.415,156.665
C08155=1046.118,58.232,417.576,170.276,35.414,156.664
C08156=1046.111,57.983,417.593,170.274,35.412,156.664
C08157=1046.105,57.734,417.610,170.272,35.410,156.664
C08158=1046.099,57.484,417.628,170.270,35.409,156.664
C08159=1046.092,57.235,417.646,170.268,35.408,156.663
C08160=1046.086,56.986,417.663,170.267,35.406,156.663
C08161=1046.079,56.737,417.681,170.265,35.405,156.663
C08162=1046.073,56.488,417.698,170.263,35.403,156.663
C08163=1046.067,56.238,417.715,170.262,35.401,156.662
C08164=1046.060,55.989,417.733,170.260,35.400,156.662
C08165=1046.055,55.739,417.750,170.258,35.399,156.662
C08166=1046.048,55.490,417.767,170.257,35.397,156.662
C08167=1046.042,55.241,417.784,170.254,35.396,156.661
C08168=1046.036,54.991,417.802,170.252,35.394,156.661
C08169=1046.029,54.742,417.819,170.251,35.392,156.661
C08170=1046.023,54.493,417.837,170.249,35.391,156.661
C08171=1046.017,54.243,417.854,170.247,35.389,156.660
C08172=1046.010,53.994,417.871,170.246,35.388,156.660
C08173=1046.004,53.744,417.888,170.244,35.387,156.660
C08174=1045.998,53.495,417.905,170.242,35.385,156.659
C08175=1045.991,53.246,417.923,170.241,35.383,156.659
C08176=1045.986,52.997,417.940,170.238,35.382,156.659
C08177=1045.979,52.747,417.958,170.236,35.380,156.659
C08178=1045.973,52.498,417.975,170.235,35.379,156.658
C08179=1045.967,52.248,417.992,170.233,35.377,156.658
C08180=1045.961,52.000,418.009,170.231,35.376,156.658
C08181=1045.955,51.750,418.027,170.230,35.374,156.658
C08182=1045.948,51.501,418.044,170.228,35.372,156.657
C08183=1045.942,51.251,418.060,170.226,35.371,156.657
C08184=1045.936,51.002,418.078,170.225,35.370,156.657
C08185=1045.929,50.753,418.095,170.222,35.368,156.657
C08186=1045.923,50.504,418.112,170.220,35.366,156.656
C08187=1045.917,50.254,418.129,170.219,35.365,156.656
C08188=1045.911,50.005,418.146,170.217,35.363,156.656
C08189=1045.904,49.755,418.164,170.215,35.362,156.656
C08190=1045.899,49.506,418.181,170.214,35.360,156.655
C08191=1045.892,49.256,418.198,170.212,35.359,156.655
C08192=1045.887,49.007,418.215,170.210,35.357,156.655
C08193=1045.880,48.758,418.233,170.209,35.356,156.654
C08194=1045.874,48.508,418.249,170.207,35.354,156.654
C08195=1045.868,48.259,418.267,170.205,35.352,156.654
C08196=1045.861,48.010,418.284,170.203,35.351,156.654
C08197=1045.855,47.761,418.301,170.201,35.350,156.653
C08198=1045.849,47.511,418.318,170.200,35.348,156.653
C08199=1045.843,47.262,418.335,170.198,35.346,156.653
C08200=1045.836,47.012,418.352,170.196,35.345,156.653
C08201=1045.831,46.763,418.369,170.195,35.343,156.652
C08202=1045.825,46.514,418.386,170.193,35.342,156.652
C08203=1045.818,46.264,418.403,170.191,35.340,156.652
C08204=1045.812,46.016,418.420,170.189,35.339,156.652
C08205=1045.806,45.767,418.437,170.187,35.337,156.651
C08206=1045.799,45.479,418.457,170.185,35.335,156.651
C08207=1045.792,45.193,418.476,170.183,35.334,156.651
C08208=1045.785,44.907,418.496,170.181,35.332,156.650
C08209=1045.777,44.620,418.515,170.179,35.330,156.650
C08210=1045.772,44.371,418.533,170.178,35.328,156.650
C08211=1045.766,44.121,418.549,170.176,35.327,156.650
C08212=1045.759,43.872,418.566,170.174,35.325,156.649
C08213=1045.753,43.623,418.583,170.172,35.324,156.649
C08214=1045.748,43.374,418.600,170.170,35.322,156.649
C08215=1045.741,43.124,418.617,170.168,35.321,156.648
C08216=1045.735,42.875,418.634,170.167,35.319,156.648
C08217=1045.728,42.625,418.650,170.165,35.318,156.648
C08218=1045.722,42.376,418.667,170.163,35.316,156.648
C08219=1045.716,42.127,418.684,170.162,35.315,156.647
C08220=1045.709,41.877,418.701,170.160,35.313,156.647
C08221=1045.703,41.628,418.717,170.158,35.312,156.647
C08222=1045.697,41.379,418.734,170.156,35.310,156.647
C08223=1045.691,41.129,418.751,170.154,35.309,156.646
C08224=1045.685,40.880,418.767,170.152,35.308,156.646
C08225=1045.678,40.631,418.784,170.150,35.306,156.646
C08226=1045.672,40.381,418.801,170.149,35.304,156.646
C08227=1045.666,40.132,418.818,170.147,35.303,156.645
C08228=1045.660,39.882,418.835,170.145,35.301,156.645
C08229=1045.654,39.633,418.851,170.144,35.300,156.645
C08230=1045.647,39.384,418.868,170.142,35.299,156.645
C08231=1045.641,39.134,418.885,170.140,35.297,156.644
C08232=1045.635,38.885,418.902,170.139,35.295,156.644
C08233=1045.629,38.636,418.918,170.136,35.294,156.644
C08234=1045.623,38.386,418.934,170.134,35.293,156.644
C08235=1045.616,38.137,418.952,170.133,35.291,156.643
C08236=1045.610,37.888,418.968,170.131,35.289,156.643
C08237=1045.604,37.638,418.984,170.129,35.288,156.643
C08238=1045.597,37.389,419.001,170.127,35.287,156.643
C08239=1045.591,37.139,419.018,170.126,35.285,156.642
C08240=1045.585,36.890,419.034,170.124,35.284,156.642
C08241=1045.579,36.640,419.051,170.122,35.282,156.642
C08242=1045.572,36.392,419.067,170.121,35.281,156.642
C08243=1045.566,36.142,419.083,170.118,35.280,156.641
C08244=1045.559,35.892,419.100,170.116,35.278,156.641
C08245=1045.553,35.643,419.116,170.114,35.276,156.641
C08246=1045.547,35.394,419.133,170.113,35.275,156.641
C08247=1045.540,35.144,419.150,170.111,35.274,156.640
C08248=1045.534,34.895,419.165,170.109,35.272,156.640
C08249=1045.528,34.646,419.182,170.108,35.271,156.640
C08250=1045.521,34.396,419.198,170.106,35.269,156.640
C08251=1045.515,34.147,419.215,170.104,35.268,156.639
C08252=1045.509,33.898,419.231,170.102,35.267,156.639
C08253=1045.503,33.648,419.248,170.101,35.265,156.639
C08254=1045.496,33.399,419.264,170.098,35.264,156.639
C08255=1045.490,33.149,419.280,170.096,35.262,156.638
C08256=1045.484,32.900,419.296,170.095,35.261,156.638
C08257=1045.478,32.651,419.312,170.093,35.259,156.638
C08258=1045.471,32.401,419.330,170.091,35.258,156.638
C08259=1045.464,32.152,419.345,170.089,35.257,156.638
C08260=1045.458,31.903,419.362,170.088,35.255,156.637
C08261=1045.452,31.653,419.378,170.086,35.254,156.637
C08262=1045.446,31.403,419.395,170.084,35.252,156.637
C08263=1045.440,31.154,419.411,170.083,35.251,156.637
C08264=1045.433,30.905,419.427,170.081,35.250,156.636
C08265=1045.427,30.656,419.443,170.078,35.248,156.636
C08266=1045.421,30.406,419.459,170.076,35.246,156.636
C08267=1045.415,30.156,419.476,170.075,35.245,156.636
C08268=1045.409,29.907,419.492,170.073,35.244,156.635
C08269=1045.402,29.658,419.508,170.071,35.242,156.635
C08270=1045.396,29.371,419.527,170.069,35.240,156.635
C08271=1045.388,29.085,419.545,170.067,35.239,156.635
C08272=1045.381,28.799,419.564,170.065,35.237,156.634
C08273=1045.373,28.512,419.583,170.063,35.235,156.634
C08274=1045.367,28.263,419.599,170.062,35.234,156.634
C08275=1045.361,28.013,419.616,170.059,35.233,156.634
C08276=1045.354,27.763,419.631,170.057,35.231,156.633
C08277=1045.349,27.514,419.647,170.055,35.230,156.633
C08278=1045.343,27.265,419.663,170.054,35.229,156.633
C08279=1045.336,27.016,419.679,170.052,35.227,156.633
C08280=1045.329,26.766,419.695,170.050,35.225,156.632
C08281=1045.323,26.516,419.712,170.049,35.224,156.632
C08282=1045.317,26.267,419.727,170.047,35.223,156.632
C08283=1045.311,26.018,419.744,170.045,35.221,156.632
C08284=1045.304,25.769,419.759,170.043,35.220,156.631
C08285=1045.298,25.520,419.775,170.042,35.219,156.631
C08286=1045.292,25.269,419.792,170.040,35.218,156.631
C08287=1045.285,25.020,419.808,170.037,35.216,156.631
C08288=1045.279,24.770,419.823,170.035,35.214,156.630
C08289=1045.273,24.521,419.839,170.034,35.213,156.630
C08290=1045.267,24.272,419.855,170.032,35.212,156.630
C08291=1045.260,24.023,419.871,170.030,35.210,156.630
C08292=1045.253,23.773,419.887,170.028,35.209,156.630
C08293=1045.247,23.524,419.903,170.027,35.208,156.629
C08294=1045.241,23.274,419.919,170.025,35.206,156.629
C08295=1045.235,23.025,419.935,170.023,35.205,156.629
C08296=1045.228,22.776,419.951,170.021,35.204,156.629
C08297=1045.222,22.526,419.967,170.020,35.202,156.628
C08298=1045.216,22.277,419.983,170.017,35.200,156.628
C08299=1045.210,22.027,419.998,170.015,35.199,156.628
C08300=1045.203,21.778,420.014,170.013,35.198,156.628
C08301=1045.197,21.528,420.030,170.012,35.197,156.628
C08302=1045.190,21.279,420.046,170.010,35.195,156.627
C08303=1045.184,21.030,420.062,170.008,35.194,156.627
C08304=1045.179,20.780,420.078,170.006,35.193,156.627
C08305=1045.172,20.531,420.093,170.005,35.191,156.627
C08306=1045.166,20.281,420.110,170.003,35.189,156.626
C08307=1045.160,20.032,420.125,170.001,35.188,156.626
C08308=1045.154,19.782,420.141,169.999,35.187,156.626
C08309=1045.147,19.533,420.157,169.997,35.185,156.626
C08310=1045.140,19.284,420.172,169.995,35.184,156.625
C08311=1045.135,19.034,420.188,169.993,35.183,156.625
C08312=1045.128,18.785,420.203,169.991,35.181,156.625
C08313=1045.122,18.535,420.219,169.989,35.180,156.625
C08314=1045.115,18.286,420.235,169.988,35.179,156.625
C08315=1045.109,18.036,420.251,169.986,35.177,156.624
C08316=1045.103,17.787,420.266,169.984,35.176,156.624
C08317=1045.096,17.538,420.282,169.982,35.175,156.624
C08318=1045.090,17.288,420.298,169.980,35.173,156.624
C08319=1045.084,17.039,420.313,169.979,35.172,156.624
C08320=1045.078,16.789,420.329,169.977,35.171,156.623
C08321=1045.071,16.540,420.344,169.975,35.170,156.623
C08322=1045.065,16.291,420.360,169.972,35.168,156.623
C08323=1045.059,16.041,420.376,169.971,35.166,156.623
C08324=1045.052,15.792,420.391,169.969,35.165,156.622
C08325=1045.046,15.542,420.407,169.967,35.164,156.622
C08326=1045.040,15.293,420.422,169.965,35.162,156.622
C08327=1045.033,15.043,420.438,169.963,35.161,156.622
C08328=1045.028,14.794,420.454,169.962,35.160,156.621
C08329=1045.021,14.544,420.469,169.960,35.158,156.621
C08330=1045.014,14.295,420.484,169.958,35.157,156.621
C08331=1045.009,14.045,420.500,169.956,35.156,156.621
C08332=1045.002,13.796,420.515,169.955,35.154,156.621
C08333=1044.995,13.547,420.531,169.953,35.153,156.620
C08334=1044.988,13.253,420.549,169.951,35.152,156.620
C08335=1044.981,12.960,420.567,169.947,35.150,156.620
C08336=1044.972,12.667,420.585,169.945,35.148,156.620
C08337=1044.965,12.373,420.604,169.943,35.147,156.619
C08338=1044.959,12.124,420.618,169.941,35.146,156.619
C08339=1044.952,11.875,420.634,169.940,35.144,156.619
C08340=1044.946,11.625,420.650,169.938,35.143,156.619
C08341=1044.940,11.375,420.665,169.936,35.142,156.619
C08342=1044.933,11.126,420.680,169.934,35.141,156.618
C08343=1044.927,10.876,420.695,169.932,35.140,156.618
C08344=1044.920,10.627,420.711,169.930,35.138,156.618
C08345=1044.914,10.378,420.726,169.929,35.137,156.618
C08346=1044.908,10.129,420.740,169.927,35.136,156.618
C08347=1044.902,9.879,420.757,169.925,35.134,156.617
C08348=1044.896,9.630,420.772,169.922,35.133,156.617
C08349=1044.889,9.380,420.787,169.920,35.132,156.617
C08350=1044.882,9.131,420.802,169.919,35.130,156.617
C08351=1044.876,8.881,420.817,169.917,35.129,156.617
C08352=1044.870,8.632,420.832,169.915,35.128,156.616
C08353=1044.863,8.383,420.848,169.913,35.126,156.616
C08354=1044.857,8.133,420.863,169.911,35.126,156.616
C08355=1044.850,7.883,420.878,169.909,35.124,156.616
C08356=1044.845,7.633,420.893,169.908,35.123,156.616
C08357=1044.838,7.384,420.909,169.906,35.122,156.615
C08358=1044.832,7.135,420.924,169.904,35.120,156.615
C08359=1044.825,6.885,420.939,169.902,35.119,156.615
C08360=1044.819,6.635,420.954,169.900,35.118,156.615
C08361=1044.813,6.387,420.969,169.898,35.116,156.615
C08362=1044.806,6.137,420.984,169.896,35.115,156.614
C08363=1044.800,5.888,420.999,169.894,35.114,156.614
C08364=1044.794,5.638,421.014,169.892,35.113,156.614
C08365=1044.788,5.389,421.030,169.890,35.111,156.614
C08366=1044.781,5.139,421.045,169.888,35.110,156.613
C08367=1044.775,4.889,421.060,169.887,35.109,156.613
C08368=1044.768,4.640,421.075,169.885,35.108,156.613
C08369=1044.763,4.391,421.089,169.883,35.107,156.613
C08370=1044.756,4.142,421.105,169.881,35.105,156.613
C08371=1044.750,3.892,421.120,169.879,35.104,156.612
C08372=1044.743,3.643,421.135,169.877,35.102,156.612
C08373=1044.737,3.393,421.150,169.875,35.101,156.612
C08374=1044.730,3.143,421.165,169.874,35.100,156.612
C08375=1044.725,2.894,421.180,169.872,35.099,156.612
C08376=1044.718,2.645,421.194,169.869,35.097,156.611
C08377=1044.712,2.395,421.211,169.867,35.096,156.611
C08378=1044.706,2.150,421.225,169.865,35.095,156.611
C08379=1044.700,1.904,421.239,169.864,35.093,156.611
C08380=1044.694,1.659,421.255,169.862,35.093,156.611
C08381=1044.687,1.413,421.269,169.860,35.091,156.610
C08382=1044.681,1.168,421.284,169.858,35.090,156.610
C08383=1044.675,0.922,421.299,169.856,35.089,156.610
C08384=1044.670,0.677,421.313,169.854,35.087,156.610
C08385=1044.663,0.432,421.328,169.853,35.086,156.610
C08386=1044.656,0.182,421.343,169.851,35.085,156.609
C08387=1044.650,-0.067,421.358,169.849,35.083,156.609
C08388=1044.644,-0.316,421.372,169.847,35.082,156.609
C08389=1044.638,-0.566,421.387,169.845,35.081,156.609
C08390=1044.632,-0.816,421.403,169.842,35.079,156.609
C08391=1044.626,-1.066,421.418,169.841,35.078,156.608
C08392=1044.620,-1.315,421.432,169.839,35.077,156.608
C08393=1044.614,-1.564,421.447,169.837,35.076,156.608
C08394=1044.607,-1.814,421.462,169.835,35.074,156.608
C08395=1044.601,-2.064,421.477,169.833,35.073,156.608
C08396=1044.595,-2.313,421.492,169.831,35.072,156.607
C08397=1044.589,-2.562,421.507,169.829,35.070,156.607
C08398=1044.582,-2.846,421.523,169.827,35.069,156.607
C08399=1044.574,-3.129,421.540,169.825,35.068,156.607
C08400=1044.568,-3.412,421.557,169.823,35.066,156.606
C08401=1044.561,-3.695,421.574,169.821,35.064,156.606
C08402=1044.553,-3.945,421.588,169.819,35.064,156.606
C08403=1044.547,-4.195,421.603,169.817,35.062,156.606
C08404=1044.542,-4.444,421.617,169.815,35.061,156.606
C08405=1044.535,-4.693,421.632,169.812,35.060,156.605
C08406=1044.528,-4.943,421.647,169.810,35.059,156.605
C08407=1044.522,-5.192,421.661,169.809,35.058,156.605
C08408=1044.516,-5.441,421.676,169.807,35.056,156.605
C08409=1044.510,-5.692,421.690,169.805,35.055,156.605
C08410=1044.503,-5.941,421.705,169.803,35.054,156.605
C08411=1044.496,-6.191,421.720,169.801,35.053,156.604
C08412=1044.491,-6.440,421.734,169.799,35.052,156.604
C08413=1044.483,-6.689,421.749,169.797,35.050,156.604
C08414=1044.477,-6.939,421.763,169.795,35.050,156.604
C08415=1044.472,-7.188,421.777,169.793,35.048,156.604
C08416=1044.465,-7.438,421.792,169.791,35.047,156.603
C08417=1044.458,-7.687,421.807,169.790,35.046,156.603
C08418=1044.453,-7.937,421.821,169.788,35.045,156.603
C08419=1044.446,-8.186,421.835,169.786,35.044,156.603
C08420=1044.439,-8.436,421.850,169.784,35.042,156.603
C08421=1044.433,-8.685,421.864,169.781,35.042,156.603
C08422=1044.427,-8.935,421.879,169.779,35.040,156.602
C08423=1044.421,-9.185,421.894,169.777,35.039,156.602
C08424=1044.414,-9.433,421.908,169.775,35.038,156.602
C08425=1044.408,-9.684,421.922,169.773,35.037,156.602
C08426=1044.402,-9.933,421.937,169.771,35.035,156.602
C08427=1044.395,-10.182,421.951,169.769,35.034,156.602
C08428=1044.389,-10.432,421.965,169.767,35.033,156.601
C08429=1044.383,-10.682,421.980,169.766,35.032,156.601
C08430=1044.376,-10.930,421.994,169.764,35.031,156.601
C08431=1044.370,-11.181,422.008,169.762,35.029,156.601
C08432=1044.364,-11.430,422.023,169.760,35.029,156.601
C08433=1044.357,-11.679,422.037,169.758,35.027,156.600
C08434=1044.351,-11.929,422.051,169.756,35.026,156.600
C08435=1044.346,-12.178,422.066,169.754,35.025,156.600
C08436=1044.339,-12.428,422.081,169.752,35.024,156.600
C08437=1044.333,-12.677,422.094,169.750,35.023,156.600
C08438=1044.327,-12.927,422.109,169.747,35.021,156.600
C08439=1044.320,-13.177,422.123,169.745,35.020,156.599
C08440=1044.314,-13.426,422.137,169.743,35.019,156.599
C08441=1044.308,-13.676,422.151,169.741,35.018,156.599
C08442=1044.302,-13.925,422.166,169.740,35.017,156.599
C08443=1044.295,-14.174,422.180,169.738,35.016,156.599
C08444=1044.290,-14.424,422.194,169.736,35.015,156.598
C08445=1044.283,-14.674,422.209,169.734,35.013,156.598
C08446=1044.276,-14.924,422.223,169.732,35.012,156.598
C08447=1044.271,-15.173,422.237,169.730,35.011,156.598
C08448=1044.264,-15.422,422.251,169.728,35.010,156.598
C08449=1044.258,-15.671,422.266,169.726,35.008,156.598
C08450=1044.251,-15.921,422.279,169.724,35.008,156.597
C08451=1044.245,-16.170,422.294,169.722,35.006,156.597
C08452=1044.239,-16.420,422.307,169.720,35.006,156.597
C08453=1044.232,-16.671,422.322,169.718,35.004,156.597
C08454=1044.226,-16.919,422.336,169.716,35.004,156.597
C08455=1044.219,-17.169,422.349,169.714,35.002,156.597
C08456=1044.213,-17.418,422.364,169.711,35.001,156.596
C08457=1044.207,-17.668,422.378,169.709,35.000,156.596
C08458=1044.201,-17.918,422.391,169.707,34.999,156.596
C08459=1044.194,-18.167,422.406,169.705,34.998,156.596
C08460=1044.188,-18.417,422.420,169.703,34.997,156.596
C08461=1044.181,-18.666,422.434,169.701,34.996,156.596
C08462=1044.174,-18.948,422.449,169.699,34.995,156.596
C08463=1044.167,-19.230,422.465,169.697,34.993,156.595
C08464=1044.160,-19.511,422.481,169.695,34.992,156.595
C08465=1044.153,-19.793,422.496,169.692,34.991,156.595
C08466=1044.146,-20.042,422.511,169.690,34.990,156.595
C08467=1044.140,-20.292,422.524,169.688,34.989,156.595
C08468=1044.134,-20.542,422.538,169.686,34.988,156.595
C08469=1044.128,-20.791,422.553,169.685,34.987,156.594
C08470=1044.121,-21.041,422.566,169.683,34.986,156.594
C08471=1044.115,-21.290,422.580,169.681,34.984,156.594
C08472=1044.108,-21.540,422.595,169.679,34.984,156.594
C08473=1044.102,-21.789,422.608,169.677,34.982,156.594
C08474=1044.097,-22.039,422.622,169.675,34.981,156.593
C08475=1044.090,-22.289,422.635,169.673,34.980,156.593
C08476=1044.083,-22.537,422.649,169.670,34.979,156.593
C08477=1044.077,-22.788,422.663,169.668,34.978,156.593
C08478=1044.071,-23.037,422.677,169.666,34.977,156.593
C08479=1044.065,-23.287,422.691,169.664,34.976,156.593
C08480=1044.059,-23.536,422.705,169.662,34.975,156.593
C08481=1044.052,-23.785,422.718,169.660,34.974,156.592
C08482=1044.046,-24.035,422.732,169.658,34.973,156.592
C08483=1044.040,-24.285,422.746,169.656,34.971,156.592
C08484=1044.033,-24.534,422.759,169.654,34.971,156.592
C08485=1044.028,-24.784,422.773,169.652,34.969,156.592
C08486=1044.021,-25.033,422.787,169.650,34.969,156.592
C08487=1044.015,-25.283,422.801,169.648,34.967,156.591
C08488=1044.009,-25.532,422.815,169.646,34.967,156.591
C08489=1044.002,-25.782,422.828,169.644,34.965,156.591
C08490=1043.997,-26.032,422.842,169.642,34.965,156.591
C08491=1043.990,-26.281,422.856,169.640,34.963,156.591
C08492=1043.983,-26.530,422.870,169.638,34.962,156.591
C08493=1043.978,-26.780,422.884,169.636,34.961,156.591
C08494=1043.972,-27.029,422.897,169.634,34.960,156.590
C08495=1043.965,-27.279,422.911,169.632,34.959,156.590
C08496=1043.959,-27.528,422.924,169.630,34.958,156.590
C08497=1043.952,-27.778,422.938,169.627,34.957,156.590
C08498=1043.946,-28.028,422.951,169.625,34.956,156.590
C08499=1043.940,-28.277,422.965,169.622,34.956,156.590
C08500=1043.933,-28.527,422.978,169.620,34.954,156.590
C08501=1043.927,-28.777,422.992,169.618,34.953,156.589
C08502=1043.920,-29.026,423.005,169.616,34.952,156.589
C08503=1043.914,-29.276,423.018,169.614,34.951,156.589
C08504=1043.908,-29.525,423.032,169.612,34.951,156.589
C08505=1043.901,-29.775,423.045,169.610,34.949,156.589
C08506=1043.895,-30.024,423.059,169.608,34.949,156.589
C08507=1043.889,-30.274,423.073,169.606,34.948,156.589
C08508=1043.882,-30.524,423.086,169.604,34.947,156.588
C08509=1043.876,-30.773,423.099,169.602,34.946,156.588
C08510=1043.870,-31.022,423.113,169.600,34.944,156.588
C08511=1043.863,-31.272,423.126,169.598,34.944,156.588
C08512=1043.857,-31.522,423.140,169.596,34.943,156.588
C08513=1043.851,-31.771,423.152,169.594,34.942,156.588
C08514=1043.844,-32.021,423.166,169.592,34.941,156.588
C08515=1043.838,-32.271,423.179,169.590,34.940,156.588
C08516=1043.832,-32.520,423.192,169.588,34.939,156.587
C08517=1043.826,-32.769,423.206,169.586,34.938,156.587
C08518=1043.820,-33.019,423.220,169.584,34.937,156.587
C08519=1043.813,-33.269,423.233,169.582,34.936,156.587
C08520=1043.807,-33.518,423.246,169.579,34.935,156.587
C08521=1043.800,-33.768,423.260,169.576,34.934,156.587
C08522=1043.794,-34.018,423.273,169.574,34.933,156.587
C08523=1043.788,-34.267,423.286,169.572,34.933,156.586
C08524=1043.782,-34.516,423.299,169.570,34.931,156.586
C08525=1043.775,-34.766,423.313,169.568,34.930,156.586
C08526=1043.768,-35.047,423.327,169.566,34.929,156.586
C08527=1043.761,-35.328,423.343,169.564,34.928,156.586
C08528=1043.754,-35.608,423.357,169.561,34.927,156.586
C08529=1043.748,-35.890,423.372,169.559,34.926,156.586
C08530=1043.742,-36.139,423.386,169.557,34.926,156.585
C08531=1043.735,-36.388,423.399,169.555,34.924,156.585
C08532=1043.729,-36.639,423.412,169.553,34.923,156.585
C08533=1043.723,-36.888,423.425,169.551,34.922,156.585
C08534=1043.716,-37.138,423.438,169.549,34.921,156.585
C08535=1043.710,-37.387,423.452,169.546,34.921,156.585
C08536=1043.704,-37.637,423.464,169.544,34.919,156.585
C08537=1043.697,-37.887,423.478,169.542,34.919,156.585
C08538=1043.691,-38.136,423.491,169.540,34.918,156.584
C08539=1043.685,-38.385,423.504,169.538,34.916,156.584
C08540=1043.679,-38.635,423.517,169.536,34.916,156.584
C08541=1043.673,-38.884,423.530,169.534,34.915,156.584
C08542=1043.666,-39.135,423.543,169.532,34.914,156.584
C08543=1043.660,-39.384,423.556,169.530,34.914,156.584
C08544=1043.654,-39.633,423.570,169.528,34.912,156.584
C08545=1043.647,-39.883,423.582,169.526,34.912,156.584
C08546=1043.641,-40.132,423.595,169.523,34.911,156.583
C08547=1043.635,-40.382,423.608,169.521,34.910,156.583
C08548=1043.628,-40.632,423.621,169.519,34.909,156.583
C08549=1043.622,-40.881,423.634,169.516,34.908,156.583
C08550=1043.616,-41.131,423.646,169.514,34.907,156.583
C08551=1043.609,-41.380,423.660,169.512,34.907,156.583
C08552=1043.603,-41.630,423.672,169.510,34.906,156.583
C08553=1043.597,-41.879,423.685,169.508,34.905,156.583
C08554=1043.590,-42.129,423.699,169.506,34.904,156.583
C08555=1043.584,-42.379,423.711,169.503,34.903,156.582
C08556=1043.578,-42.628,423.724,169.501,34.902,156.582
C08557=1043.572,-42.878,423.737,169.499,34.901,156.582
C08558=1043.565,-43.127,423.750,169.497,34.901,156.582
C08559=1043.560,-43.377,423.763,169.495,34.900,156.582
C08560=1043.553,-43.626,423.775,169.493,34.899,156.582
C08561=1043.546,-43.877,423.788,169.491,34.899,156.582
C08562=1043.540,-44.126,423.801,169.489,34.897,156.582
C08563=1043.534,-44.376,423.814,169.486,34.896,156.582
C08564=1043.528,-44.625,423.827,169.484,34.896,156.581
C08565=1043.521,-44.875,423.839,169.482,34.895,156.581
C08566=1043.515,-45.125,423.852,169.480,34.894,156.581
C08567=1043.509,-45.374,423.865,169.478,34.894,156.581
C08568=1043.503,-45.624,423.878,169.476,34.893,156.581
C08569=1043.496,-45.873,423.890,169.474,34.892,156.581
C08570=1043.490,-46.123,423.903,169.472,34.891,156.581
C08571=1043.484,-46.372,423.916,169.469,34.890,156.581
C08572=1043.478,-46.622,423.929,169.467,34.889,156.581
C08573=1043.471,-46.871,423.941,169.465,34.889,156.581
C08574=1043.465,-47.121,423.954,169.463,34.888,156.580
C08575=1043.459,-47.370,423.966,169.461,34.887,156.580
C08576=1043.453,-47.620,423.979,169.459,34.886,156.580
C08577=1043.447,-47.870,423.993,169.457,34.885,156.580
C08578=1043.440,-48.120,424.005,169.454,34.884,156.580
C08579=1043.434,-48.369,424.018,169.452,34.884,156.580
C08580=1043.428,-48.619,424.030,169.450,34.883,156.580
C08581=1043.421,-48.869,424.042,169.448,34.882,156.580
C08582=1043.415,-49.119,424.055,169.446,34.881,156.580
C08583=1043.409,-49.368,424.068,169.443,34.881,156.579
C08584=1043.403,-49.618,424.081,169.441,34.880,156.579
C08585=1043.397,-49.867,424.092,169.438,34.879,156.579
C08586=1043.390,-50.117,424.106,169.436,34.878,156.579
C08587=1043.384,-50.366,424.119,169.434,34.877,156.579
C08588=1043.378,-50.616,424.131,169.432,34.876,156.579
C08589=1043.372,-50.866,424.143,169.430,34.876,156.579
C08590=1043.365,-51.147,424.157,169.427,34.875,156.579
C08591=1043.357,-51.428,424.171,169.425,34.874,156.579
C08592=1043.350,-51.710,424.185,169.422,34.873,156.579
C08593=1043.343,-51.990,424.199,169.420,34.873,156.578
C08594=1043.336,-52.240,424.211,169.418,34.873,156.579
C08595=1043.331,-52.490,424.223,169.415,34.872,156.578
C08596=1043.324,-52.739,424.235,169.413,34.871,156.578
C08597=1043.318,-52.989,424.248,169.411,34.870,156.578
C08598=1043.311,-53.238,424.260,169.409,34.870,156.578
C08599=1043.304,-53.488,424.272,169.407,34.869,156.578
C08600=1043.299,-53.738,424.285,169.404,34.868,156.578
C08601=1043.292,-53.987,424.297,169.402,34.868,156.578
C08602=1043.286,-54.237,424.309,169.400,34.867,156.578
C08603=1043.279,-54.487,424.321,169.398,34.867,156.578
C08604=1043.273,-54.736,424.333,169.396,34.866,156.578
C08605=1043.267,-54.986,424.346,169.393,34.865,156.578
C08606=1043.260,-55.236,424.358,169.391,34.864,156.578
C08607=1043.253,-55.485,424.370,169.389,34.864,156.577
C08608=1043.248,-55.735,424.382,169.387,34.864,156.577
C08609=1043.241,-55.985,424.394,169.385,34.863,156.577
C08610=1043.235,-56.235,424.407,169.382,34.862,156.577
C08611=1043.228,-56.484,424.419,169.380,34.861,156.577
C08612=1043.222,-56.734,424.431,169.378,34.861,156.577
C08613=1043.216,-56.984,424.443,169.376,34.860,156.577
C08614=1043.209,-57.233,424.455,169.374,34.860,156.577
C08615=1043.203,-57.482,424.467,169.371,34.859,156.577
C08616=1043.197,-57.732,424.479,169.369,34.858,156.577
C08617=1043.191,-57.982,424.491,169.367,34.858,156.577
C08618=1043.184,-58.231,424.503,169.365,34.857,156.577
C08619=1043.178,-58.481,424.516,169.362,34.857,156.577
C08620=1043.171,-58.731,424.528,169.360,34.856,156.577
C08621=1043.165,-58.981,424.540,169.358,34.855,156.577
C08622=1043.159,-59.230,424.552,169.356,34.855,156.576
C08623=1043.153,-59.479,424.564,169.354,34.854,156.576
C08624=1043.147,-59.729,424.577,169.351,34.854,156.576
C08625=1043.140,-59.978,424.589,169.349,34.853,156.576
C08626=1043.134,-60.228,424.601,169.347,34.852,156.576
C08627=1043.128,-60.478,424.613,169.345,34.851,156.576
C08628=1043.121,-60.728,424.624,169.342,34.851,156.576
C08629=1043.115,-60.978,424.636,169.340,34.851,156.576
C08630=1043.109,-61.227,424.648,169.338,34.850,156.576
C08631=1043.103,-61.476,424.660,169.336,34.849,156.576
C08632=1043.096,-61.726,424.672,169.333,34.848,156.576
C08633=1043.090,-61.976,424.685,169.331,34.848,156.576
C08634=1043.083,-62.225,424.697,169.329,34.848,156.576
C08635=1043.078,-62.475,424.708,169.327,34.847,156.576
C08636=1043.071,-62.725,424.720,169.325,34.846,156.576
C08637=1043.065,-62.974,424.732,169.322,34.845,156.575
C08638=1043.059,-63.224,424.744,169.320,34.845,156.575
C08639=1043.053,-63.473,424.756,169.318,34.845,156.575
C08640=1043.047,-63.723,424.768,169.316,34.844,156.575
C08641=1043.040,-63.973,424.780,169.313,34.843,156.575
C08642=1043.034,-64.222,424.792,169.311,34.843,156.575
C08643=1043.028,-64.472,424.804,169.309,34.842,156.575
C08644=1043.022,-64.722,424.815,169.307,34.841,156.575
C08645=1043.015,-64.971,424.827,169.303,34.841,156.575
C08646=1043.009,-65.221,424.839,169.302,34.841,156.575
C08647=1043.003,-65.470,424.851,169.299,34.840,156.575
C08648=1042.997,-65.720,424.862,169.297,34.839,156.575
C08649=1042.990,-65.970,424.874,169.294,34.838,156.575
C08650=1042.984,-66.220,424.887,169.292,34.838,156.575
C08651=1042.979,-66.469,424.898,169.290,34.838,156.575
C08652=1042.972,-66.719,424.910,169.288,34.837,156.575
C08653=1042.965,-66.968,424.922,169.285,34.836,156.574
C08654=1042.959,-67.251,424.935,169.283,34.836,156.574
C08655=1042.952,-67.534,424.948,169.280,34.835,156.574
C08656=1042.945,-67.816,424.961,169.278,34.834,156.574
C08657=1042.938,-68.099,424.974,169.275,34.834,156.574
C08658=1042.932,-68.348,424.987,169.273,34.833,156.574
C08659=1042.926,-68.599,424.998,169.271,34.833,156.574
C08660=1042.920,-68.847,425.010,169.268,34.832,156.574
C08661=1042.914,-69.097,425.022,169.266,34.831,156.574
C08662=1042.908,-69.348,425.034,169.264,34.831,156.574
C08663=1042.902,-69.596,425.045,169.262,34.831,156.574
C08664=1042.895,-69.847,425.056,169.259,34.830,156.574
C08665=1042.889,-70.097,425.069,169.257,34.830,156.574
C08666=1042.884,-70.346,425.080,169.255,34.829,156.574
C08667=1042.877,-70.596,425.092,169.253,34.828,156.574
C08668=1042.871,-70.844,425.103,169.250,34.828,156.574
C08669=1042.865,-71.095,425.115,169.248,34.827,156.574
C08670=1042.859,-71.345,425.127,169.246,34.827,156.574
C08671=1042.853,-71.594,425.138,169.243,34.826,156.573
C08672=1042.846,-71.844,425.150,169.241,34.826,156.573
C08673=1042.841,-72.093,425.161,169.239,34.825,156.573
C08674=1042.835,-72.343,425.173,169.237,34.824,156.573
C08675=1042.829,-72.592,425.184,169.234,34.824,156.573
C08676=1042.822,-72.842,425.196,169.232,34.823,156.573
C08677=1042.816,-73.092,425.208,169.230,34.823,156.573
C08678=1042.811,-73.341,425.220,169.228,34.823,156.573
C08679=1042.804,-73.592,425.231,169.225,34.822,156.573
C08680=1042.798,-73.841,425.242,169.223,34.822,156.573
C08681=1042.792,-74.091,425.254,169.221,34.821,156.573
C08682=1042.786,-74.340,425.265,169.218,34.820,156.573
C08683=1042.779,-74.590,425.277,169.216,34.820,156.573
C08684=1042.773,-74.840,425.288,169.214,34.820,156.573
C08685=1042.767,-75.089,425.299,169.212,34.819,156.573
C08686=1042.761,-75.339,425.311,169.209,34.819,156.573
C08687=1042.755,-75.588,425.322,169.207,34.818,156.573
C08688=1042.749,-75.839,425.333,169.205,34.818,156.573
C08689=1042.743,-76.087,425.344,169.202,34.818,156.573
C08690=1042.736,-76.338,425.356,169.200,34.818,156.573
C08691=1042.730,-76.588,425.367,169.198,34.817,156.573
C08692=1042.724,-76.837,425.379,169.195,34.817,156.573
C08693=1042.718,-77.087,425.390,169.193,34.816,156.573
C08694=1042.712,-77.336,425.401,169.191,34.816,156.573
C08695=1042.705,-77.587,425.412,169.188,34.816,156.573
C08696=1042.699,-77.835,425.423,169.186,34.815,156.573
C08697=1042.693,-78.086,425.435,169.184,34.815,156.573
C08698=1042.687,-78.335,425.445,169.181,34.814,156.573
C08699=1042.680,-78.585,425.456,169.179,34.814,156.573
C08700=1042.674,-78.834,425.468,169.177,34.813,156.572
C08701=1042.668,-79.084,425.479,169.174,34.813,156.573
C08702=1042.662,-79.334,425.490,169.172,34.813,156.573
C08703=1042.656,-79.584,425.501,169.170,34.812,156.572
C08704=1042.650,-79.833,425.513,169.167,34.812,156.572
C08705=1042.643,-80.083,425.524,169.165,34.811,156.572
C08706=1042.638,-80.332,425.535,169.163,34.811,156.572
C08707=1042.631,-80.582,425.546,169.160,34.811,156.572
C08708=1042.625,-80.832,425.556,169.158,34.811,156.572
C08709=1042.619,-81.082,425.568,169.156,34.811,156.572
C08710=1042.612,-81.331,425.578,169.153,34.810,156.572
C08711=1042.606,-81.581,425.589,169.151,34.810,156.572
C08712=1042.600,-81.830,425.601,169.149,34.810,156.572
C08713=1042.593,-82.080,425.612,169.146,34.810,156.572
C08714=1042.587,-82.330,425.622,169.144,34.809,156.572
C08715=1042.580,-82.580,425.634,169.142,34.809,156.572
C08716=1042.575,-82.829,425.644,169.139,34.809,156.572
C08717=1042.568,-83.079,425.655,169.137,34.809,156.572
C08718=1042.561,-83.364,425.667,169.134,34.808,156.572
C08719=1042.553,-83.648,425.680,169.131,34.808,156.572
C08720=1042.547,-83.933,425.692,169.129,34.808,156.572
C08721=1042.539,-84.218,425.704,169.126,34.808,156.572
C08722=1042.534,-84.468,425.715,169.124,34.808,156.572
C08723=1042.527,-84.718,425.726,169.121,34.807,156.572
C08724=1042.521,-84.968,425.737,169.119,34.807,156.572
C08725=1042.514,-85.218,425.748,169.117,34.807,156.572
C08726=1042.509,-85.467,425.759,169.114,34.807,156.572
C08727=1042.503,-85.716,425.770,169.112,34.806,156.572
C08728=1042.496,-85.966,425.780,169.109,34.806,156.572
C08729=1042.490,-86.216,425.791,169.107,34.806,156.572
C08730=1042.484,-86.465,425.802,169.105,34.806,156.572
C08731=1042.477,-86.715,425.813,169.102,34.805,156.572
C08732=1042.472,-86.965,425.824,169.100,34.805,156.573
C08733=1042.464,-87.215,425.834,169.098,34.805,156.573
C08734=1042.459,-87.464,425.845,169.095,34.804,156.572
C08735=1042.453,-87.714,425.856,169.093,34.804,156.572
C08736=1042.446,-87.963,425.867,169.091,34.804,156.573
C08737=1042.440,-88.214,425.877,169.089,34.804,156.573
C08738=1042.435,-88.463,425.888,169.087,34.804,156.573
C08739=1042.428,-88.713,425.898,169.084,34.804,156.573
C08740=1042.422,-88.962,425.909,169.082,34.804,156.573
C08741=1042.416,-89.212,425.920,169.080,34.803,156.573
C08742=1042.409,-89.462,425.931,169.077,34.803,156.573
C08743=1042.403,-89.711,425.942,169.075,34.803,156.573
C08744=1042.398,-89.961,425.952,169.072,34.803,156.573
C08745=1042.391,-90.211,425.962,169.070,34.803,156.573
C08746=1042.385,-90.461,425.973,169.068,34.803,156.573
C08747=1042.379,-90.710,425.984,169.065,34.802,156.573
C08748=1042.373,-90.959,425.994,169.063,34.802,156.573
C08749=1042.367,-91.210,426.005,169.060,34.802,156.573
C08750=1042.360,-91.459,426.015,169.058,34.801,156.573
C08751=1042.355,-91.709,426.026,169.056,34.801,156.573
C08752=1042.348,-91.958,426.036,169.053,34.801,156.573
C08753=1042.342,-92.208,426.048,169.051,34.801,156.573
C08754=1042.336,-92.458,426.058,169.049,34.801,156.573
C08755=1042.330,-92.708,426.068,169.046,34.801,156.573
C08756=1042.324,-92.957,426.079,169.044,34.801,156.573
C08757=1042.317,-93.207,426.090,169.041,34.801,156.573
C08758=1042.312,-93.457,426.100,169.039,34.801,156.573
C08759=1042.306,-93.707,426.111,169.037,34.800,156.573
C08760=1042.299,-93.956,426.121,169.034,34.800,156.573
C08761=1042.293,-94.207,426.132,169.032,34.800,156.573
C08762=1042.287,-94.456,426.142,169.029,34.799,156.573
C08763=1042.281,-94.705,426.153,169.027,34.799,156.573
C08764=1042.276,-94.955,426.163,169.025,34.799,156.573
C08765=1042.269,-95.204,426.173,169.022,34.799,156.573
C08766=1042.264,-95.454,426.184,169.020,34.799,156.573
C08767=1042.257,-95.704,426.194,169.017,34.799,156.573
C08768=1042.251,-95.954,426.205,169.015,34.799,156.573
C08769=1042.245,-96.203,426.215,169.013,34.799,156.573
C08770=1042.239,-96.453,426.225,169.010,34.799,156.573
C08771=1042.233,-96.703,426.236,169.008,34.799,156.573
C08772=1042.227,-96.953,426.246,169.005,34.798,156.573
C08773=1042.221,-97.203,426.257,169.003,34.798,156.573
C08774=1042.215,-97.453,426.266,169.001,34.798,156.573
C08775=1042.209,-97.702,426.277,168.998,34.798,156.573
C08776=1042.202,-97.951,426.288,168.996,34.798,156.573
C08777=1042.196,-98.201,426.297,168.993,34.798,156.573
C08778=1042.191,-98.450,426.308,168.991,34.798,156.573
C08779=1042.184,-98.701,426.318,168.988,34.798,156.573
C08780=1042.177,-98.950,426.328,168.986,34.798,156.573
C08781=1042.172,-99.200,426.338,168.984,34.798,156.573
C08782=1042.165,-99.488,426.350,168.981,34.798,156.573
C08783=1042.157,-99.774,426.362,168.978,34.798,156.573
C08784=1042.150,-100.062,426.374,168.975,34.798,156.574
C08785=1042.143,-100.348,426.385,168.972,34.798,156.574
C08786=1042.137,-100.598,426.395,168.970,34.798,156.574
C08787=1042.131,-100.849,426.405,168.967,34.798,156.574
C08788=1042.125,-101.098,426.415,168.965,34.798,156.574
C08789=1042.118,-101.347,426.425,168.963,34.798,156.574
C08790=1042.113,-101.597,426.436,168.960,34.798,156.574
C08791=1042.107,-101.847,426.445,168.958,34.798,156.574
C08792=1042.100,-102.097,426.455,168.955,34.798,156.574
C08793=1042.095,-102.346,426.466,168.953,34.798,156.574
C08794=1042.088,-102.596,426.475,168.951,34.798,156.574
C08795=1042.082,-102.845,426.486,168.949,34.798,156.574
C08796=1042.076,-103.095,426.495,168.947,34.798,156.574
C08797=1042.070,-103.345,426.505,168.944,34.798,156.574
C08798=1042.063,-103.595,426.516,168.942,34.799,156.574
C08799=1042.057,-103.845,426.526,168.939,34.799,156.574
C08800=1042.052,-104.095,426.536,168.937,34.798,156.574
C08801=1042.045,-104.344,426.546,168.934,34.798,156.574
C08802=1042.039,-104.594,426.556,168.932,34.799,156.575
C08803=1042.033,-104.844,426.565,168.929,34.799,156.575
C08804=1042.027,-105.094,426.575,168.927,34.799,156.575
C08805=1042.021,-105.343,426.586,168.924,34.799,156.575
C08806=1042.015,-105.593,426.595,168.922,34.799,156.575
C08807=1042.009,-105.842,426.605,168.920,34.799,156.575
C08808=1042.003,-106.093,426.615,168.917,34.799,156.575
C08809=1041.997,-106.342,426.625,168.915,34.799,156.575
C08810=1041.991,-106.591,426.635,168.912,34.799,156.575
C08811=1041.984,-106.841,426.644,168.910,34.799,156.575
C08812=1041.978,-107.091,426.654,168.907,34.799,156.575
C08813=1041.972,-107.341,426.665,168.905,34.800,156.575
C08814=1041.966,-107.590,426.674,168.902,34.799,156.575
C08815=1041.960,-107.840,426.684,168.900,34.800,156.575
C08816=1041.954,-108.090,426.694,168.897,34.800,156.575
C08817=1041.948,-108.340,426.703,168.895,34.800,156.575
C08818=1041.942,-108.590,426.713,168.892,34.800,156.576
C08819=1041.935,-108.839,426.722,168.890,34.800,156.576
C08820=1041.929,-109.089,426.733,168.887,34.801,156.576
C08821=1041.923,-109.338,426.742,168.885,34.801,156.576
C08822=1041.917,-109.588,426.752,168.883,34.801,156.576
C08823=1041.911,-109.838,426.762,168.880,34.801,156.576
C08824=1041.905,-110.088,426.771,168.878,34.801,156.576
C08825=1041.899,-110.338,426.781,168.875,34.801,156.576
C08826=1041.893,-110.588,426.791,168.873,34.801,156.576
C08827=1041.887,-110.837,426.800,168.871,34.802,156.576
C08828=1041.881,-111.087,426.809,168.869,34.802,156.576
C08829=1041.875,-111.336,426.819,168.866,34.802,156.576
C08830=1041.869,-111.586,426.828,168.864,34.802,156.576
C08831=1041.862,-111.836,426.838,168.861,34.803,156.577
C08832=1041.856,-112.086,426.848,168.859,34.803,156.577
C08833=1041.850,-112.335,426.858,168.856,34.803,156.577
C08834=1041.844,-112.585,426.867,168.854,34.803,156.577
C08835=1041.837,-112.834,426.877,168.851,34.804,156.577
C08836=1041.832,-113.085,426.887,168.849,34.804,156.577
C08837=1041.826,-113.334,426.897,168.846,34.804,156.577
C08838=1041.821,-113.584,426.905,168.844,34.804,156.577
C08839=1041.814,-113.834,426.915,168.841,34.804,156.577
C08840=1041.808,-114.084,426.924,168.839,34.804,156.577
C08841=1041.802,-114.334,426.934,168.836,34.805,156.577
C08842=1041.796,-114.583,426.944,168.834,34.805,156.577
C08843=1041.790,-114.833,426.953,168.831,34.805,156.578
C08844=1041.784,-115.083,426.963,168.829,34.805,156.578
C08845=1041.777,-115.333,426.972,168.826,34.806,156.578
C08846=1041.771,-115.618,426.982,168.823,34.806,156.578
C08847=1041.763,-115.904,426.994,168.821,34.806,156.578
C08848=1041.756,-116.191,427.004,168.818,34.807,156.578
C08849=1041.749,-116.477,427.015,168.815,34.807,156.578
C08850=1041.743,-116.727,427.024,168.812,34.807,156.578
C08851=1041.738,-116.976,427.034,168.810,34.808,156.578
C08852=1041.731,-117.226,427.043,168.807,34.808,156.578
C08853=1041.726,-117.476,427.052,168.805,34.808,156.578
C08854=1041.719,-117.726,427.062,168.803,34.809,156.579
C08855=1041.712,-117.976,427.071,168.801,34.809,156.579
C08856=1041.706,-118.225,427.080,168.798,34.809,156.579
C08857=1041.701,-118.474,427.089,168.796,34.809,156.579
C08858=1041.695,-118.725,427.098,168.793,34.810,156.579
C08859=1041.689,-118.975,427.108,168.791,34.810,156.579
C08860=1041.683,-119.224,427.117,168.788,34.810,156.579
C08861=1041.676,-119.474,427.127,168.786,34.811,156.579
C08862=1041.670,-119.723,427.135,168.783,34.811,156.579
C08863=1041.664,-119.973,427.144,168.781,34.811,156.579
C08864=1041.658,-120.223,427.154,168.778,34.812,156.580
C08865=1041.652,-120.473,427.163,168.776,34.812,156.580
C08866=1041.647,-120.723,427.172,168.773,34.812,156.580
C08867=1041.640,-120.973,427.182,168.771,34.813,156.580
C08868=1041.634,-121.222,427.191,168.768,34.813,156.580
C08869=1041.627,-121.472,427.200,168.766,34.813,156.580
C08870=1041.622,-121.722,427.209,168.763,34.814,156.580
C08871=1041.616,-121.971,427.218,168.761,34.814,156.580
C08872=1041.610,-122.221,427.228,168.758,34.815,156.581
C08873=1041.604,-122.472,427.237,168.756,34.815,156.581
C08874=1041.598,-122.720,427.245,168.753,34.815,156.581
C08875=1041.591,-122.970,427.255,168.751,34.816,156.581
C08876=1041.585,-123.221,427.264,168.748,34.816,156.581
C08877=1041.580,-123.470,427.273,168.746,34.817,156.581
C08878=1041.574,-123.720,427.282,168.744,34.817,156.581
C08879=1041.567,-123.970,427.291,168.741,34.817,156.581
C08880=1041.562,-124.219,427.300,168.739,34.818,156.581
C08881=1041.556,-124.469,427.309,168.736,34.818,156.582
C08882=1041.550,-124.719,427.318,168.734,34.819,156.582
C08883=1041.543,-124.969,427.326,168.731,34.820,156.582
C08884=1041.537,-125.218,427.336,168.729,34.819,156.582
C08885=1041.532,-125.469,427.345,168.726,34.820,156.582
C08886=1041.525,-125.718,427.353,168.724,34.821,156.582
C08887=1041.519,-125.968,427.362,168.721,34.821,156.582
C08888=1041.513,-126.218,427.372,168.719,34.822,156.582
C08889=1041.507,-126.468,427.380,168.716,34.822,156.583
C08890=1041.501,-126.717,427.389,168.714,34.823,156.583
C08891=1041.495,-126.967,427.398,168.711,34.823,156.583
C08892=1041.488,-127.217,427.407,168.708,34.824,156.583
C08893=1041.483,-127.466,427.415,168.706,34.824,156.583
C08894=1041.477,-127.716,427.425,168.703,34.825,156.583
C08895=1041.471,-127.965,427.434,168.701,34.825,156.583
C08896=1041.467,-128.215,427.443,168.699,34.825,156.583
C08897=1041.463,-128.465,427.454,168.696,34.824,156.583
C08898=1041.459,-128.715,427.465,168.694,34.823,156.583
C08899=1041.457,-128.965,427.476,168.692,34.821,156.583
C08900=1041.455,-129.215,427.489,168.691,34.820,156.583
C08901=1041.454,-129.465,427.501,168.689,34.817,156.582
C08902=1041.454,-129.715,427.515,168.687,34.814,156.582
C08903=1041.456,-129.965,427.528,168.686,34.810,156.581
C08904=1041.458,-130.215,427.543,168.685,34.807,156.581
C08905=1041.461,-130.465,427.558,168.683,34.802,156.580
C08906=1041.464,-130.716,427.573,168.682,34.798,156.579
C08907=1041.468,-130.966,427.590,168.681,34.793,156.578
C08908=1041.473,-131.216,427.607,168.680,34.787,156.577
C08909=1041.480,-131.466,427.624,168.679,34.781,156.576
C08910=1041.131,-131.490,427.370,168.631,34.973,156.610
C08911=1041.125,-131.240,427.351,168.633,34.979,156.611
C08912=1041.120,-130.990,427.335,168.634,34.985,156.611
C08913=1041.115,-130.739,427.318,168.634,34.990,156.612
C08914=1041.112,-130.489,427.303,168.636,34.995,156.613
C08915=1041.109,-130.240,427.287,168.638,34.999,156.614
C08916=1041.108,-129.989,427.272,168.639,35.003,156.615
C08917=1041.106,-129.739,427.259,168.640,35.006,156.615
C08918=1041.106,-129.489,427.245,168.642,35.009,156.615
C08919=1041.107,-129.239,427.233,168.643,35.012,156.616
C08920=1041.108,-128.989,427.220,168.646,35.014,156.616
C08921=1041.111,-128.739,427.209,168.648,35.015,156.616
C08922=1041.114,-128.489,427.198,168.650,35.016,156.617
C08923=1041.118,-128.239,427.187,168.652,35.017,156.617
C08924=1041.122,-127.989,427.178,168.655,35.017,156.617
C08925=1041.128,-127.740,427.168,168.657,35.017,156.617
C08926=1041.134,-127.491,427.160,168.660,35.016,156.616
C08927=1041.140,-127.241,427.151,168.661,35.016,156.616
C08928=1041.146,-126.991,427.141,168.664,35.015,156.616
C08929=1041.152,-126.742,427.134,168.666,35.014,156.616
C08930=1041.158,-126.492,427.124,168.669,35.014,156.616
C08931=1041.164,-126.241,427.115,168.671,35.014,156.616
C08932=1041.170,-125.993,427.107,168.674,35.013,156.616
C08933=1041.176,-125.742,427.098,168.677,35.013,156.616
C08934=1041.183,-125.492,427.088,168.679,35.012,156.615
C08935=1041.189,-125.243,427.080,168.682,35.012,156.615
C08936=1041.195,-124.993,427.071,168.684,35.011,156.615
C08937=1041.201,-124.743,427.062,168.687,35.011,156.615
C08938=1041.207,-124.494,427.053,168.689,35.010,156.615
C08939=1041.213,-124.244,427.044,168.692,35.010,156.615
C08940=1041.219,-123.994,427.035,168.694,35.009,156.615
C08941=1041.225,-123.743,427.026,168.697,35.009,156.615
C08942=1041.230,-123.494,427.017,168.699,35.009,156.614
C08943=1041.237,-123.245,427.008,168.702,35.008,156.614
C08944=1041.243,-122.994,426.999,168.705,35.008,156.614
C08945=1041.249,-122.745,426.990,168.707,35.007,156.614
C08946=1041.255,-122.495,426.980,168.710,35.006,156.614
C08947=1041.261,-122.245,426.971,168.712,35.007,156.614
C08948=1041.268,-121.995,426.962,168.714,35.006,156.614
C08949=1041.273,-121.746,426.953,168.716,35.005,156.614
C08950=1041.279,-121.496,426.944,168.719,35.005,156.614
C08951=1041.285,-121.246,426.935,168.721,35.004,156.613
C08952=1041.291,-120.997,426.925,168.724,35.004,156.613
C08953=1041.297,-120.747,426.917,168.726,35.004,156.613
C08954=1041.304,-120.497,426.908,168.729,35.003,156.613
C08955=1041.310,-120.247,426.898,168.731,35.003,156.613
C08956=1041.315,-119.998,426.890,168.734,35.003,156.613
C08957=1041.321,-119.748,426.880,168.736,35.002,156.613
C08958=1041.327,-119.498,426.870,168.739,35.002,156.613
C08959=1041.334,-119.248,426.861,168.742,35.001,156.613
C08960=1041.340,-118.998,426.853,168.744,35.001,156.612
C08961=1041.346,-118.749,426.843,168.747,35.001,156.612
C08962=1041.352,-118.499,426.834,168.749,35.000,156.612
C08963=1041.358,-118.249,426.824,168.752,35.000,156.612
C08964=1041.364,-118.000,426.815,168.754,35.000,156.612
C08965=1041.370,-117.749,426.806,168.757,34.999,156.612
C08966=1041.376,-117.500,426.797,168.759,34.999,156.612
C08967=1041.382,-117.250,426.787,168.762,34.999,156.612
C08968=1041.388,-117.001,426.778,168.764,34.998,156.612
C08969=1041.394,-116.751,426.768,168.767,34.998,156.612
C08970=1041.401,-116.501,426.760,168.769,34.998,156.611
C08971=1041.407,-116.215,426.749,168.771,34.997,156.611
C08972=1041.414,-115.929,426.738,168.774,34.997,156.611
C08973=1041.421,-115.642,426.727,168.777,34.997,156.611
C08974=1041.428,-115.357,426.716,168.780,34.996,156.611
C08975=1041.434,-115.106,426.707,168.782,34.996,156.611
C08976=1041.440,-114.856,426.697,168.785,34.996,156.611
C08977=1041.447,-114.606,426.688,168.787,34.995,156.611
C08978=1041.452,-114.357,426.679,168.790,34.995,156.611
C08979=1041.458,-114.108,426.669,168.792,34.995,156.611
C08980=1041.464,-113.858,426.659,168.795,34.994,156.610
C08981=1041.471,-113.608,426.650,168.797,34.994,156.610
C08982=1041.477,-113.358,426.640,168.800,34.994,156.610
C08983=1041.483,-113.108,426.631,168.802,34.994,156.610
C08984=1041.489,-112.859,426.621,168.805,34.993,156.610
C08985=1041.495,-112.609,426.612,168.807,34.994,156.610
C08986=1041.501,-112.360,426.602,168.810,34.993,156.610
C08987=1041.507,-112.110,426.593,168.812,34.993,156.610
C08988=1041.513,-111.860,426.583,168.815,34.993,156.610
C08989=1041.519,-111.610,426.574,168.817,34.993,156.610
C08990=1041.526,-111.361,426.564,168.820,34.992,156.610
C08991=1041.532,-111.111,426.555,168.822,34.992,156.610
C08992=1041.538,-110.861,426.545,168.825,34.992,156.609
C08993=1041.544,-110.611,426.535,168.827,34.992,156.609
C08994=1041.550,-110.361,426.525,168.830,34.991,156.609
C08995=1041.556,-110.111,426.516,168.832,34.991,156.609
C08996=1041.562,-109.861,426.506,168.835,34.991,156.609
C08997=1041.568,-109.612,426.497,168.837,34.991,156.609
C08998=1041.575,-109.362,426.486,168.839,34.990,156.609
C08999=1041.581,-109.113,426.477,168.841,34.990,156.609
C09000=1041.587,-108.863,426.467,168.844,34.990,156.609
C09001=1041.593,-108.613,426.458,168.846,34.990,156.609
C09002=1041.599,-108.363,426.448,168.849,34.989,156.609
C09003=1041.605,-108.113,426.438,168.851,34.989,156.609
C09004=1041.612,-107.864,426.429,168.854,34.989,156.609
C09005=1041.618,-107.614,426.419,168.856,34.989,156.609
C09006=1041.623,-107.364,426.408,168.859,34.989,156.608
C09007=1041.629,-107.115,426.399,168.861,34.989,156.608
C09008=1041.635,-106.865,426.390,168.864,34.989,156.608
C09009=1041.641,-106.616,426.380,168.866,34.988,156.608
C09010=1041.648,-106.367,426.370,168.869,34.988,156.608
C09011=1041.653,-106.116,426.360,168.871,34.988,156.608
C09012=1041.659,-105.867,426.350,168.874,34.988,156.608
C09013=1041.666,-105.616,426.340,168.876,34.988,156.608
C09014=1041.673,-105.367,426.330,168.879,34.988,156.608
C09015=1041.678,-105.117,426.320,168.881,34.987,156.608
C09016=1041.684,-104.867,426.310,168.883,34.988,156.608
C09017=1041.691,-104.617,426.301,168.886,34.988,156.608
C09018=1041.697,-104.368,426.290,168.888,34.987,156.608
C09019=1041.702,-104.118,426.280,168.891,34.987,156.608
C09020=1041.709,-103.868,426.271,168.893,34.987,156.608
C09021=1041.715,-103.619,426.260,168.896,34.987,156.608
C09022=1041.721,-103.369,426.251,168.898,34.987,156.607
C09023=1041.727,-103.119,426.241,168.901,34.987,156.607
C09024=1041.733,-102.870,426.230,168.903,34.987,156.607
C09025=1041.739,-102.620,426.221,168.906,34.987,156.607
C09026=1041.745,-102.370,426.211,168.908,34.987,156.607
C09027=1041.751,-102.121,426.200,168.911,34.987,156.607
C09028=1041.757,-101.871,426.191,168.913,34.987,156.607
C09029=1041.763,-101.621,426.181,168.915,34.986,156.607
C09030=1041.769,-101.372,426.170,168.918,34.986,156.607
C09031=1041.776,-101.121,426.160,168.920,34.986,156.607
C09032=1041.782,-100.872,426.149,168.922,34.987,156.607
C09033=1041.788,-100.622,426.140,168.924,34.987,156.607
C09034=1041.794,-100.373,426.130,168.927,34.986,156.607
C09035=1041.802,-100.085,426.118,168.930,34.986,156.607
C09036=1041.808,-99.798,426.107,168.932,34.986,156.607
C09037=1041.816,-99.511,426.095,168.935,34.986,156.607
C09038=1041.822,-99.224,426.083,168.938,34.986,156.607
C09039=1041.829,-98.974,426.073,168.940,34.986,156.607
C09040=1041.835,-98.724,426.063,168.943,34.986,156.607
C09041=1041.841,-98.474,426.053,168.945,34.986,156.607
C09042=1041.847,-98.225,426.042,168.948,34.986,156.607
C09043=1041.853,-97.975,426.033,168.950,34.986,156.606
C09044=1041.859,-97.726,426.022,168.953,34.986,156.606
C09045=1041.866,-97.475,426.012,168.955,34.986,156.606
C09046=1041.872,-97.226,426.002,168.958,34.986,156.606
C09047=1041.878,-96.977,425.991,168.960,34.986,156.606
C09048=1041.883,-96.727,425.981,168.962,34.986,156.606
C09049=1041.890,-96.477,425.970,168.965,34.986,156.606
C09050=1041.895,-96.227,425.960,168.967,34.986,156.606
C09051=1041.902,-95.978,425.950,168.970,34.987,156.606
C09052=1041.908,-95.728,425.939,168.972,34.987,156.606
C09053=1041.914,-95.478,425.929,168.974,34.987,156.606
C09054=1041.920,-95.229,425.918,168.977,34.987,156.606
C09055=1041.926,-94.979,425.907,168.979,34.987,156.606
C09056=1041.932,-94.729,425.898,168.982,34.987,156.606
C09057=1041.938,-94.479,425.887,168.984,34.987,156.606
C09058=1041.945,-94.230,425.876,168.986,34.987,156.606
C09059=1041.950,-93.980,425.866,168.989,34.987,156.606
C09060=1041.956,-93.730,425.855,168.991,34.987,156.606
C09061=1041.962,-93.481,425.845,168.994,34.988,156.606
C09062=1041.969,-93.230,425.835,168.996,34.988,156.606
C09063=1041.975,-92.981,425.824,168.998,34.988,156.606
C09064=1041.981,-92.732,425.813,169.001,34.988,156.606
C09065=1041.986,-92.482,425.803,169.003,34.988,156.606
C09066=1041.993,-92.232,425.793,169.006,34.988,156.606
C09067=1041.999,-91.982,425.782,169.008,34.988,156.606
C09068=1042.005,-91.733,425.771,169.011,34.988,156.606
C09069=1042.011,-91.484,425.761,169.013,34.988,156.606
C09070=1042.017,-91.233,425.750,169.015,34.988,156.606
C09071=1042.024,-90.984,425.740,169.018,34.989,156.606
C09072=1042.029,-90.734,425.729,169.020,34.989,156.606
C09073=1042.036,-90.485,425.719,169.023,34.989,156.606
C09074=1042.042,-90.235,425.707,169.025,34.989,156.606
C09075=1042.048,-89.985,425.697,169.027,34.990,156.606
C09076=1042.054,-89.735,425.687,169.030,34.990,156.606
C09077=1042.061,-89.485,425.676,169.032,34.990,156.606
C09078=1042.066,-89.236,425.665,169.034,34.990,156.606
C09079=1042.073,-88.987,425.654,169.037,34.990,156.606
C09080=1042.079,-88.736,425.643,169.039,34.990,156.606
C09081=1042.085,-88.487,425.634,169.042,34.990,156.606
C09082=1042.091,-88.237,425.623,169.044,34.990,156.606
C09083=1042.097,-87.987,425.612,169.046,34.990,156.606
C09084=1042.104,-87.738,425.601,169.049,34.991,156.606
C09085=1042.110,-87.488,425.590,169.051,34.991,156.606
C09086=1042.116,-87.238,425.579,169.054,34.991,156.606
C09087=1042.122,-86.989,425.569,169.056,34.991,156.606
C09088=1042.128,-86.739,425.558,169.058,34.991,156.606
C09089=1042.134,-86.489,425.547,169.061,34.992,156.606
C09090=1042.141,-86.240,425.536,169.063,34.992,156.606
C09091=1042.147,-85.991,425.526,169.066,34.992,156.606
C09092=1042.153,-85.740,425.514,169.068,34.992,156.606
C09093=1042.159,-85.491,425.504,169.070,34.993,156.606
C09094=1042.166,-85.240,425.494,169.073,34.993,156.606
C09095=1042.171,-84.991,425.483,169.075,34.993,156.606
C09096=1042.178,-84.742,425.472,169.077,34.993,156.606
C09097=1042.184,-84.492,425.461,169.079,34.993,156.605
C09098=1042.190,-84.242,425.450,169.081,34.993,156.605
C09099=1042.197,-83.957,425.437,169.085,34.994,156.606
C09100=1042.204,-83.673,425.425,169.087,34.994,156.606
C09101=1042.211,-83.387,425.413,169.089,34.994,156.606
C09102=1042.219,-83.103,425.400,169.092,34.994,156.605
C09103=1042.225,-82.853,425.389,169.094,34.994,156.605
C09104=1042.231,-82.604,425.379,169.097,34.995,156.606
C09105=1042.238,-82.354,425.368,169.099,34.995,156.606
C09106=1042.243,-82.104,425.357,169.102,34.995,156.605
